(* CODESYS project devicelib.library
   Author: AMKO-Engineering
   Placeholder: Device_Library
   Title: Device_Library
   Version: 1.2.0.3
   Description: Device library of AMKO-Engineering.
   Company: AMKO-Engineering

Project tree, tasks and I/O mapping:
  libraries: HMI_Library, * (AMKO-Engineering); Tc2_MC2, * (Beckhoff Automation GmbH); Tc2_MC2_Drive, * (Beckhoff Automation GmbH); Tc2_Standard, * (Beckhoff Automation GmbH); Utilities_Library, * (AMKO-Engineering)
  Actuators/
    Cylinder/
      DataTypes/
        ManualControls/
          data type UDT_ManualValveControl
        data type E_CylinderCmd
        data type E_ValveResetState
      Functions/
        function block Fb_DevCylWithFbk [ST]: CalcTimers, ExecDirection, ExecSetFeedback, ExecTimeout, CmdSimulate, CmdTeach, Init
        function block FB_DevValve [ST]: ExecSetFeedback, ExecSetOutPuts, CmdClose, CmdHold, CmdManual, CmdOpen, CmdReset, CmdSafeStop, CmdTeach, Init
      MLTFunctions/
        function block Fb_DevSupportCyl [ST]: ExecCalc, ExecCylControl, ExecFaultHandling, Init_Support, Mod_ManualControl, Mod_SupportDown
  Axis/
    DataTypes/
      data type E_AxisCmd
      data type UDT_AxisData
      data type UDT_AxVal
    FunctionBlocks/
      function block Fb_DevAxis [ST]: CmdGearDynamic, CmdGearIn, CmdGearOut, CmdHalt, CmdHome, CmdJog, CmdLimitVelocity, CmdManual, CmdMoveAbs, CmdMoveModulo, CmdMoveRelative, CmdMoveVelocity, CmdReset, CmdSafeSpeed, CmdSafeStop, Init, ExecGearDynamic, ExecGearIn, ExecGearOut, ExecHalt, ExecHome, ExecJog, ExecMoveAbsolute, ExecMoveModulo, ExecMoveRelative, ExecMoveVelocity, ExecEnable, ExecReadStatus, ExecReset, ExecSafeFunctions, CallMotionFunctions, CallOrganizationFunctions
      function block FB_DevBasicACAxis [ST]: CmdHalt, CmdHome, CmdJog, CmdManual, CmdMoveAbs, CmdMoveRelative, CmdMoveVelocity, CmdReset, CmdSafeStop, Init, ExecEnable, ExecHalt, ExecHome, ExecJog, ExecMoveAbsolute, ExecMoveRelative, ExecMoveVelocity, ExecReset, ExecSafeFunctions, CallMotionFunctions
      function block FB_DevHybridAc [ST]: ExecHalt, ExecReadStatus, ExecReset, Init
      data type UDT_ManualAxisCtrl
    Interface/
  BaseFunctions/
    function block FB_DevBase [ST]: ExecIdentifyDevice, CalcDeviceId, CmdManual, CmdReset, CmdSafeStop, ExecMessagTest
    data type UDT_DevManualCtrl
  Buttons/
    DataTypes/
    Functions/
      function block FB_DevHMIButton [ST]
      function block FB_DevPushButton [ST]
      function block FB_DevPushbuttonLight [ST]: CmdBlinkFast, CmdBlinkSlow, CmdOn
  DevTypes/
    data type E_Devices
  Encoders/
    DataTypes/
    FunctionBlocks/
      function block FB_EncoderBase [ST]: FastTask
      function block FB_EncoderInput [ST]: FastTask
  GroupHandlers/
    ManualControlHandler/
      function block FB_ManualController [ST]: ExecSelectDevice, CmdAddDevice
      data type UDT_DeviceID
    global variables GVL_DevManual
  HardwareDiagnostics/
    function block FB_ELModuleDiag [ST]
  Heaters/
    function block FB_DevDoublePWM [ST]: CalcCycleTimes, ExecPWMCycle, SetOutputs, CmdHold, CmdOutputAOn, CmdOutputBOn, CmdSafeStop, Init
    function block FB_DevPWMGenerator [ST]: CalcCycle, ExecSetOutput, CmdOutputCycle, CmdOutputOff, CmdOutputOn
  Lights/
    DataTypes/
    Functions/
      function block Fb_DevLight [ST]: ExecSetOutput, CmdBlinkFast, CmdBlinkSlow, CmdOn
  Outputs/
    AnalogOutputs/
      function block FB_DevAnalogOutput [ST]: ExecSetFeedback, ExecSetOutput
      function block FB_DevAnalogOutputScaled [ST]: ExecSetFeedback, ExecSetOutput, SetScaling
    DigitalOutputs/
      function block FB_DevDigitalOutput [ST]: ExecSetFeedback, ExecSetOutput
  Sensors/
    AnalogInput/
      FunctionBlocks/
        function block FB_DevAnalogInAutoCalibrate [ST]: CmdCalibrateNull, CmdCalilbrateValue
        function block FB_DevAnalogInput [ST]: ExecSetFeedback
        function block FB_DevAnalogInputScaled [ST]: ExecSetFeedback, SetScaling
        function block FB_DevHDAnalogInAutoCalibrate [ST]: CmdCalibrateNull, CmdCalilbrateValue
        function block FB_DevHDAnalogInput [ST]: ExecSetFeedback
        function block FB_DevHDAnalogInputScaled [ST]: ExecSetFeedback, SetScaling
    DigitalSensor/
      DataTypes/
      FunctionBlocks/
        function block Fb_DevDigitalInput [ST]
        function block Fb_DevDigitalInputFunctions [ST]
    FootPedals/
      DataTypes/
        data type E_FootpedalPos
      FunctionBlocks/
        function block FB_EfkaEB301A_FootPedal [ST]: ACT_ConvertGreycode, ACT_CreateEdges
    ModuleSpecific/
      EL3556_Loadcell/
        function block Fb_DevEL3356_LoadCell [ST]: CheckELSignalState, CmdCalibrateNull, CmdCalilbrateValue
  Version/
    global variables Global_Version
*)

// Actuators/Cylinder/DataTypes/ManualControls/UDT_ManualValveControl
TYPE UDT_ManualValveControl extends UDT_DevManualCtrl:
STRUCT
	// Device commands
	bCmdOpen	: BOOL	; // open valve 
	bCmdClose	: BOOL	; // Close valve
	bCmdTeach	: BOOL	; // Teach valve
END_STRUCT
END_TYPE

// Actuators/Cylinder/DataTypes/E_CylinderCmd
(* cylinder commands *)
TYPE E_CylinderCmd :
(
	Cyl_Idle 		:= 0,// Jog Cylinder command Referance 0 Idle (wait for command)
	Cyl_Init 		:= 1,// Jog Cylinder command Referance 1 initialize Cylinder
	Cyl_Enable 		:= 2,// Jog Cylinder command Referance 2 enable
	Cyl_Disable 	:= 3,// Jog Cylinder command Referance 3 disable
	Cyl_Reset 		:= 4,// Jog Cylinder command Referance 4 reset
	Cyl_Hold 		:= 5,// Jog Cylinder command Referance 5 hold
	Cyl_Teach 		:= 6,// Jog Cylinder command Referance 6 teach timeout settings
	Cyl_Calculate 	:= 7,// Jog Cylinder command Referance 7 calculate timeout settings from parameters
	Cyl_Expand 		:= 8,// Jog Cylinder command Referance 8 expand
	Cyl_Retract 	:= 9 // Jog Cylinder command Referance 9 retract
);
END_TYPE

// Actuators/Cylinder/DataTypes/E_ValveResetState
{attribute 'qualified_only'}
{attribute 'strict'}
TYPE E_ValveResetState :
(
	Res_Idle 		:= 0,
	Res_Closed		:= 1,
	Res_Open		:= 2
);
END_TYPE

// Axis/DataTypes/E_AxisCmd
(* axis command structure *)
TYPE E_AxisCmd :
(
	Ax_Idle 		:= 0,// Axis command Referance 0 Axis Idle
	Ax_Init 		:= 1,// Axis command Referance 1 Initialize axis
	Ax_Enable 		:= 2,// Axis command Referance 2 Enable
	Ax_Disable 		:= 3,// Axis command Referance 3 Disable
	Ax_Reset 		:= 4,// Axis command Referance 4 Reset
	Ax_Hold 		:= 5,// Axis command Referance 5 Hold
	Ax_Home 		:= 6,// Axis command Referance 6 Home
	Ax_JogFwd 		:= 7,// Axis command Referance 7 Jog Forward
	Ax_JogRev 		:= 8,// Axis command Referance 8 Jog Reverse
	Ax_MoveRelative := 9,// Axis command Referance 9 Move axis relative
	Ax_MoveAbs 		:= 10,// Axis command Referance 11 Move absolute reverse
	Ax_MoveModulo 	:= 11,// Axis command Referance 11 Move Module
	Ax_MoveVeloFwd 	:= 12,// Axis command Referance 12 Move velocity forward
	Ax_MoveVeloRev 	:= 13,// Axis command Referance 13 Move velocity reverse
	Ax_HardStop 	:= 14,// Axis command Referance 14 hard stop or emergency stop
	Ax_SoftStop 	:= 15,// Axis command Referance 15 soft stop after motion command
	Ax_GearSlave 	:= 16,// Axis command Referance 16 gear axis as slave
	Ax_GearSlaveDyn	:= 17,// Axis command Referance 17 gear axis as slave dynamic
	Ax_GearOutSlave := 18,// Axis command Referance 18 gear out from Master axis 
	Ax_Maintenance	:= 50 // Axis Command referance 50 maintenance mode, axis enabled with no command active
);
END_TYPE

// Axis/DataTypes/UDT_AxisData
TYPE UDT_AxisData:
STRUCT
	// ===== Axis name =====
		AxisName	: STRING 	; // Name of the axis (used for fault handling and identification)
		AxisNumber	: INT		; // Axis number 

	// ===== Fault data =====
		Message			: UDT_Fault 	; // Message data from Cylinder
		MessageActive	: BOOL			; // Message is active
		ErrorActive 	: BOOL 			;	// Axis in error state

	// ===== Axis Commands =====
		// ***** Enable command	*****
			CmdEnable		: BOOL 		; // Command enable axis
		// ***** Active commands *****
			AxisCmd			: E_AxisCmd ; // Axis command
			AxisSafeCmd		: E_AxisCmd	; // Axis safe command
			AxisAct			: E_AxisCmd ; // Axis Active status
		// ***** Command Modes *****
			CmdHomingMode 	: MC_HomingMode ; // Homing Mode ( MC_DefaultHoming, MC_Direct, MC_ForceCallibration, MC_ResetCallibration)
			CmdJogMode		: E_JogMode 	;
			CmdBuffermode	: MC_BufferMode	; // Buffermode used for command transition 	 
	// ===== Axis Safe commands =====
		SafeCmdLimitVelo: BOOL 	; // safe command limit velocity
		SafeCmdVelocity	: LREAL ; // Safe command velocity
		SafeCmdStop		: BOOL 	; // Stop command from safety or collision detection		
		SafeVeloLimit	: LREAL ; // safe velocity limit (link to FPAR)
	// ===== Status indication active =====
		ActHoming	: BOOL ; // Axis is homing
		ActBusy		: BOOL ; // Axis is Busy 
		ActMoving	: BOOL ; // Axis is moving
		ActAtVelo	: BOOL ; // Axis is at command velocity (only when written in Move velocity mode)

	// ===== Status indication done  =====
		FcoInit		: BOOL ; // Axis is initialised
		FcoIdle		: BOOL ; // Axis is idle enable required
		FcoEnabled	: BOOL ; // Axis is enabled
		FcoHomed	: BOOL ; // Axis is homed
		FcoGeared	: BOOL ; // Axis is geared to master axis
		FcoHeld		: BOOL ; // Axis is holding
		FcoStopped	: BOOL ; // Axis is stopped
		FcoReset	: BOOL ; // Axis reset done
		FcoReady 	: BOOL ; // Axis is ready for command
		FcoAtCmdPos	: BOOL ; // Axis is at command position (tol 0.2 deg)
		FcoCmdActive: BOOL ; // Axis new command values are active
		
	// ===== Move values =====
		Pos			: UDT_Axval	; // possition values (0 = infinite)
		Velocity 	: UDT_AxVal	; // Velocity values
		Accel		: UDT_Axval ; // Aceleration values
		Decel		: UDT_Axval ; // Deceleration values
		Torque		: UDT_Axval ; // Torque values
		EncTurnoverVal	: DINT 	; // Encoder turnover value
		TimeDisableDelay : TIME ; // Time off delay after axis move command (remove enable)
		
	// ===== Config Bits =====
		IcfCommandSpeedRpm	: BOOL ; // input speeds in Rpm
		IcfEnableForward 	: BOOL ; // Enable forward motion
 		IcfEnablereverse	: BOOL ; // Enable reverse motion
		IcfContinuous		: BOOL ; // continuous motion possible (no endpoint)
		IcfAlwaysEnable		: BOOL ; // 1 = Axis always enabled, 0 = Axis disabled at Idle 
		
	// ===== Master Axis =====
		MasterAxisRef	: REFERENCE TO AXIS_REF ; // Master axis reference (if applicable)
		GearMasterRev	: UINT	:= 1	; // Master Axis Gearing revolutions (Denominator)
		GearSlaveRev	: LREAL	:= 1	; // Slave Axis gearing revolutions (numerator)	
		ReverseSlave	: BOOL 	; // Reverse slave axis relative to master
		 
END_STRUCT
END_TYPE

// Axis/DataTypes/UDT_AxVal
TYPE UDT_AxVal :
STRUCT
	// ***** Velocity settings *****
		HardMax		: LREAL 	; // Hardware maximum set absolute maximum
		ManMax 		: LREAL		; // Manual maximum percentage of hardware max
		AutoMax		: LREAL		; // Automatic maximum percentage of hardware max
		HomeMax		: LREAL 	; // Homing maximum percentage of hardware max
		CmdVal		: LREAL 	; // Commanded value
		SafeVal		: LREAL		; // Command value after safety check
		PrevVal		: LREAL		; // previous command value 
		ActVal		: LREAL		; // Actual value
		ActModulo	: LREAL		; // [deg] Modulo position
		RefVal		: LREAL 	; // referance value (basic setting or home) 
END_STRUCT
END_TYPE

// Axis/FunctionBlocks/UDT_ManualAxisCtrl
TYPE UDT_ManualAxisCtrl :
STRUCT
	bCmdJogForward	: 	BOOL 		; // command jog forward
	bCmdJogReverse	: 	BOOL 		; // command jog reverse
	bCmdInching		: 	BOOL 		; // Command move relative Distance
	bCmdToPos		: 	BOOL 		; // command move to absolute position (only moving when active)
	bCmdHome		: 	BOOL 		; // Command home axis
	fPosition		:	LREAL 		; // target position
	fDistance		:	LREAL 		; // target position
	fVelocity		: 	LREAL 		; // Maximum velocity [units/sec]
END_STRUCT
END_TYPE

// BaseFunctions/UDT_DevManualCtrl
TYPE UDT_DevManualCtrl :
STRUCT
END_STRUCT
END_TYPE

// DevTypes/E_Devices
{attribute 'qualified_only'}
{attribute 'strict'}
{attribute 'To String'}
TYPE E_Devices :
(
	Undefined,
	Valve,
	Cylinder,
	Axis,
	PushButtonLight,
	DigitalSensor,
	AnalogSensor,
	DigitalOut,
	AnalogOut,
	PWMController,
	DoublePWMController	
)INT;
END_TYPE

// GroupHandlers/ManualControlHandler/UDT_DeviceID
TYPE UDT_DeviceID :
STRUCT
	sName			: STRING	; // device name
	sType			: STRING	; // Type of device [string for visu]
	pFunction		: POINTER TO FB_DevBase ; // Pointer to the device
END_STRUCT
END_TYPE

// Sensors/FootPedals/DataTypes/E_FootpedalPos
{attribute 'qualified_only'}
{attribute 'strict'}
TYPE E_FootpedalPos :
(
	eReverse2 	,
	eReverse1 	,
	eIdle		,
	eForward1	,
	eForward2	,
	eForward3	,
	eForward4	,
	eForward5	,
	eForward6	,
	eForward7	,
	eForward8	,
	eForward9	,
	eForward10	,
	eForward11	,
	eForward12	,
	eForward13	,
	eFalse			
) INT; 
END_TYPE

// GroupHandlers/GVL_DevManual
{attribute 'qualified_only'}
VAR_GLOBAL
	fbManualControler	: FB_ManualController ; // Default Manual control function for devices (not called implicitly) 
	bManualModeActive	: BOOL ; // System manual mode is active
END_VAR
VAR_GLOBAL CONSTANT
	nMAXDEVCOUNT		: UDINT  := 100		; // Maximum number of devices 
END_VAR

// Version/Global_Version
{attribute 'TcGenerated'}
{attribute 'no-analysis'}
{attribute 'linkalways'}
// This function has been automatically generated from the project information.
VAR_GLOBAL CONSTANT
	{attribute 'const_non_replaced'}
	stLibVersion_Device_Library : ST_LibVersion := (iMajor := 1, iMinor := 2, iBuild := 0, iRevision := 3, nFlags := 0, sVersion := '1.2.0.3');
END_VAR

// Actuators/Cylinder/Functions/Fb_DevCylWithFbk
FUNCTION_BLOCK PUBLIC Fb_DevCylWithFbk EXTENDS FB_DevValve
VAR_INPUT
	bIcfFbkOpenPresent 	: BOOL := FALSE ; // Feedback for cylinder open is present 
	bIcfFbkClosedPresent: BOOL := FALSE ; // Feedback for Cylinder closed is present
	bIcfTimeChecked		: BOOL := TRUE 	; // Cylinder timing is checked = default true
	nMargin				: LREAL:= 10	; // % of tollerance in move speed 
END_VAR
VAR_OUTPUT
	// ===== Teach function =======
	bCmdCopyTimeParam 	: BOOL	:= FALSE 	;// Cylinder, Command to higher level copy toucht time to parameters
	bFeClosed			: BOOL 	:= FALSE	; // closed sensor falling edge
	bReClosed			: BOOL 	:= FALSE	; // closed sensor rising edge
	bFeOpen				: BOOL 	:= FALSE 	; // Open sensor falling edge
	bReOpen				: BOOL 	:= false 	; // open sensor rising edge 
END_VAR
VAR	
	bFcoCalcDone	: BOOL := FALSE ; // Calculate timers done 
	
	stTimesClose	: Udt_TimerBandwith ; // Timer bandwith for cylinder close
	stTimesOpen		: Udt_TimerBandwith	; // Timer bandwitch for cylinder open 
	
	fbSensorClosed	: Fb_DevDigitalInputFunctions ; // Digital sensor function closed detection
	fbSensorOpen	: Fb_DevDigitalInputFunctions ; // Digital sensor function open detection
	
	fbTimerOpen		: TON ; // Timer for cylinder to open
	fbTimerClose 	: TON ; // Timer for cylinder to close
	fbTimerTeach	: TON ; // timer for teachin cylinder 

	rtCmdWriteParam	: R_TRIG ; // Write parameter rising edge trigger 
	// Simulation
	fbTimerSimOpen 	: TON 	; 
	fbTimerSimClose	: TON 	; 
	
	// Time Cylinder valid 
	bTriggerTimeClose	: BOOL ;
	bTriggerTimeOpen	: BOOL ;
END_VAR

// set device type
	IF eDevType = E_Devices.Undefined THEN 
		eDevType := E_Devices.Cylinder ;
	END_IF

// call base function 
	SUPER^();

// check for device init
	IF NOT bInitOk THEN
		RETURN;
	END_IF 

// ====== Check direction of movement =======
	ExecDirection();
	
// ====== Check movement speed =======
	ExecTimeout();
	
// ====== Calculate timers =======
	CalcTimers();

METHOD PRIVATE CalcTimers : BOOL
VAR
END_VAR
IF stParTimeToClose.fValue = stTimesClose.Nominal AND stParTimeToOpen.fValue = stTimesOpen.Nominal AND bFcoCalcDone THEN 
	RETURN ;
ELSE
	bFcoCalcDone := FALSE ;
END_IF
 
// ====== Calculate close times ======
	stTimesClose.Nominal 	:= stParTimeToClose.fValue ;
	stTimesClose.Maximum 	:= stParTimeToClose.fValue * (1 + (nMargin / 100));
	stTimesClose.Minimal 	:= stParTimeToClose.fValue * (1 - (nMargin / 100));

// ====== Calculate open times ======
	stTimesOpen.Nominal 	:= stParTimeToOpen.fValue ;
	stTimesOpen.Maximum 	:= stParTimeToOpen.fValue * (1 + (nMargin / 100));
	stTimesOpen.Minimal 	:= stParTimeToOpen.fValue * (1 - (nMargin / 100));
	
// ====== Set feedback =======
	bFcoCalcDone := TRUE ;

// ===== send write parameters command ======	
	rtCmdWriteParam(CLK := bFcoCalcDone);
	bCmdCopyTimeParam := rtCmdWriteParam.Q	;
END_METHOD

METHOD PRIVATE ExecDirection : BOOL
VAR_INPUT
END_VAR
// ===== Check direction commands =====
 	IF q_Close AND fbSensorOpen.bReStatus AND NOT q_Open THEN
		stFault.Active			:= TRUE ;
		stFault.MessageNumber	:= E_MessageNumbers.CF_WrongDirection 	;
		stFault.Discription		:= CONCAT( sDevName,'Cylinder Opening instead of closing');
		stFault.FaultType		:= E_FaultTypes.CF 					;
		bErrorActive			:= TRUE 								;
		refFbFault.CmdAddFault( stFault );
	ELSIF q_Open AND fbSensorClosed.bReStatus AND NOT q_close THEN
		stFault.Active			:= TRUE ;
		stFault.MessageNumber	:= E_MessageNumbers.CF_WrongDirection 	;
		stFault.Discription		:= CONCAT( sDevName,'Cylinder closing instead of opening');
		stFault.FaultType		:= E_FaultTypes.CF 					;
		bErrorActive			:= TRUE 								;
	END_IF
END_METHOD

METHOD PROTECTED ExecSetFeedback : BOOL
VAR_INPUT
END_VAR
// ====== Call sensor Open function =======
	IF bIcfFbkClosedPresent THEN 
		fbSensorClosed();
		bFco_Closed := fbSensorClosed.bFcoInputActive ;
		bFeClosed 	:= fbSensorClosed.bFeStatus ;
		bReClosed 	:= fbSensorClosed.bReStatus ;
	ELSE 
		fbTOnClose	(IN 	:= q_Close, PT 	:= LREAL_TO_TIME(stParTimeToClose.fValue))	;
		bFco_Closed := fbTOnClose.Q ;
	END_IF

// ====== Call sensor Close function =======
	IF bIcfFbkOpenPresent THEN 
		fbSensorOpen() 	;
		bFco_open 	:= fbSensorOpen.bFcoInputActive ;
		bFeOpen		:= fbSensorOpen.bFeStatus;
		bReOpen		:= fbSensorOpen.bReStatus;
	ELSE 
		FbTOnOpen	(IN 	:= q_Open, PT 	:= LREAL_TO_TIME(stParTimeToOpen.fValue))	;
		bFco_Open := FbTOnOpen.Q ;
	END_IF

// ====== set outputs =======
	bReady		:= bFco_Closed OR bFco_Open ;
END_METHOD

METHOD PRIVATE ExecTimeout : BOOL
VAR_INPUT
END_VAR
VAR
	nTimePassedMs : LREAL ;
END_VAR
IF bFcoCalcDone AND bIcfTimeChecked AND bEnable THEN 
// ====== Set triggers ======
	IF q_Close  AND bFco_Open THEN 
		bTriggerTimeClose := TRUE ;
	ELSIF q_Open OR bFco_Closed  THEN 
		bTriggerTimeClose := FALSE ;
	END_IF

	IF q_Open  AND bFco_Closed THEN 
		bTriggerTimeOpen := TRUE ;
	ELSIF q_Close OR bFco_Open THEN
		bTriggerTimeOpen := FALSE ;
	END_IF
ELSE
	bTriggerTimeClose 	:= FALSE ;
	bTriggerTimeOpen	:= FALSE ;
END_IF


//======= run timers =======
	IF bIcfFbkClosedPresent THEN 
		fbTimerClose(IN := q_Close AND bEnable, PT := T#1M);
	END_IF	
	
	IF bIcfFbkOpenPresent THEN 
		fbTimerOpen	(IN := q_Open AND bEnable , PT := T#1M);
	END_IF

//====== Run timeout checks for cylinder close =======
	nTimePassedMs:= TIME_TO_LREAL(fbTimerClose.ET);
	
	IF bIcfFbkClosedPresent THEN 
		IF bTriggerTimeClose THEN 
			IF fbSensorClosed.bReStatus THEN 
				IF nTimePassedMs < stTimesClose.Minimal THEN 
					stFault.Active			:= TRUE 							;
					stFault.MessageNumber	:= E_MessageNumbers.CF_MoveToFast 	;
					stFault.Discription		:= CONCAT( sDevName,'Cylinder closing to fast')		;
					stFault.FaultType		:= E_FaultTypes.CF 					;
					bErrorActive			:= TRUE 							;
				END_IF
			ELSIF	nTimePassedMs > stTimesClose.Maximum  THEN
				stFault.Active			:= TRUE ;
				stFault.MessageNumber	:= E_MessageNumbers.CF_MoveToSlow 	;
				stFault.Discription		:= CONCAT( sDevName,'Cylinder closing to Slow')		;
				stFault.FaultType		:= E_FaultTypes.CF 				;
				bErrorActive			:= TRUE 							;
			END_IF
		END_IF
	END_IF	

//====== Run timeout checks for cylinder Open =======
	nTimePassedMs:= TIME_TO_REAL(fbTimerOpen.ET);

	IF bIcfFbkOpenPresent THEN 
		IF bTriggerTimeOpen THEN 
			IF fbSensorOpen.bReStatus THEN 
				IF nTimePassedMs < stTimesOpen.Minimal THEN 
					stFault.Active			:= TRUE ;
					stFault.MessageNumber	:= E_MessageNumbers.CF_MoveToFast 	;
					stFault.Discription		:= CONCAT( sDevName, 'Cylinder Opening to fast'	)	;
					stFault.FaultType		:= E_FaultTypes.CF 				;
					bErrorActive			:= TRUE 							;
				END_IF
			ELSIF	nTimePassedMs > stTimesOpen.Maximum  THEN
				stFault.Active			:= TRUE ;
				stFault.MessageNumber	:= E_MessageNumbers.CF_MoveToSlow 	;
				stFault.Discription		:= CONCAT( sDevName,'Cylinder Opening to Slow')		;
				stFault.FaultType		:= E_FaultTypes.CF 				;
				bErrorActive			:= TRUE 							;
			END_IF
		END_IF
	END_IF	

// Handle faults 
IF stFault.Active THEN 
	refFbFault.CmdAddFault( stFault );
END_IF
END_METHOD

METHOD PUBLIC CmdSimulate : BOOL
VAR_INPUT
	bFbkReverse		: BOOL := FALSE ; 
	tTimeSimOpen	: TIME := T#1S 	;
	tTimeSimClose	: TIME := T#1S 	;  
END_VAR
// Run timers when cylinder is active 
	fbTimerSimOpen	(IN := q_Open	, PT := tTimeSimOpen);
	fbTimerSimClose	(IN := q_Close	, PT := tTimeSimClose);

// set feedback sensors to simulate
	fbSensorOpen.bCmdSimulate 	:= TRUE ;
	fbSensorClosed.bCmdSimulate := TRUE ;

// set simulated feedback state 
	IF bFbkReverse THEN 
		fbSensorClosed.bSimState:= fbTimerSimOpen.Q 	;
		fbSensorOpen.bSimState	:= fbTimerSimClose.Q 	; 	
	ELSE 
		fbSensorClosed.bSimState:= fbTimerSimClose.Q 	;
		fbSensorOpen.bSimState	:= fbTimerSimOpen.Q 	; 	
	END_IF
END_METHOD

METHOD PUBLIC CmdTeach : BOOL
VAR_INPUT
END_VAR
// ====== turn off time check function until new calculation cycle =======
	bFcoCalcDone := false ;

// ====== teach cylinder from hardware inputs ======
	fbTimerTeach	(PT:= T#60S);
	fbTimerSwitchDir(PT:= T#1S); 
// ====== time cylinder cycles ======
	// ===== Start test loop =====
	IF bFco_Closed AND fbTimerSwitchDir.Q THEN
		bCmdClose 			:= FALSE;
		bCmdOpen 			:= TRUE ;
		fbTimerSwitchDir.IN	:= FALSE; 
		fbTimerTeach.IN 	:= TRUE ;
	ELSIF bFco_Open AND fbTimerSwitchDir.Q THEN
		bCmdClose 			:= TRUE ;
		bCmdOpen 			:= FALSE;
		fbTimerSwitchDir.IN	:= FALSE; 
		fbTimerTeach.IN 	:= TRUE ;
	ELSIF NOT bCmdClose AND NOT bCmdOpen THEN 
		bCmdClose 			:= TRUE ;
		bCmdOpen 			:= FALSE;
		fbTimerTeach.IN 	:= TRUE ;
	END_IF

// ====== start timing ========
	IF bCmdClose AND bFco_Closed THEN 
		IF fbTimerTeach.IN THEN
			stParTimeToClose.fValue 	:= TIME_TO_LREAL(fbTimerTeach.ET);
		END_IF
		fbTimerSwitchDir.IN := TRUE 		;
		fbTimerTeach.IN 	:= FALSE 		;
	ELSIF bCmdOpen AND bFco_Open THEN 
		IF fbTimerTeach.IN THEN
			stParTimeToOpen.fValue		:= TIME_TO_LREAL(fbTimerTeach.ET);
		END_IF
		fbTimerSwitchDir.IN := TRUE 		;
		fbTimerTeach.IN 	:= FALSE 		;
	END_IF
END_METHOD

METHOD PUBLIC Init : BOOL
VAR_INPUT
	// Valve data
	nDevNumber	: UDINT				:= 0		; // Cylinder identification number
	// Command state
	eResetState		: E_ValveResetState := 0		; // Cylinder reset state variable (default is idle) 
	eSafeState		: E_ValveResetState	:= 0		; // Valve safe state
END_VAR
bFcoCalcDone := FALSE;

// Enable sensor feedback
fbSensorClosed.bEnable	:= TRUE ;
fbSensorOpen.bEnable	:= TRUE ;

// Call feedback sensors 
ExecSetFeedback(); 

SUPER^.Init(nDevNumber, eResetState, eSafeState);

// ===== Set device type for manual control =====
eDevType := E_Devices.Cylinder ;


Init := bInitOk ;
END_METHOD

END_FUNCTION_BLOCK

// Actuators/Cylinder/Functions/FB_DevValve
FUNCTION_BLOCK PUBLIC FB_DevValve EXTENDS FB_DevBase
VAR_INPUT
	// Manual control 
	stManualCtrl	: UDT_ManualValveControl ;
END_VAR
VAR_OUTPUT
	// ===== Status indicators =======
	bFco_Closed		:	BOOL := FALSE ;
	bFco_Open		: 	BOOL := FALSE ;
END_VAR
VAR
	// Pararmeters
		stParTimeToClose	: Udt_Parameter := (fValue := 50) ; // time to close parameter
		stParTimeToOpen		: Udt_Parameter	:= (fValue := 50) ; // Time to open parameter
	// Hardware links 
		q_Open			AT %Q* : BOOL := FALSE 	; // Open valve
		q_Close 		AT %Q* : BOOL := FALSE	; // Close valve
	// Internal commands
		bCmdClose 	: BOOL := FALSE ; // close valve 
		bCmdOpen	: BOOL := FALSE ; // Open valve
		bCmdHold	: BOOL := FALSE ; // Hold valve status change
	// Time functions 
		fbTOnClose	: TON	; // Timer for valve close
		FbTOnOpen	: TON 	; // Timer for valve Open
		fbTimerSwitchDir: TON ; // Time for teach function switch direction 
	// reset and safe state
		eResetState		: E_ValveResetState := 0		; // Cylinder reset state variable (default is idle) 
		eSafeState		: E_ValveResetState	:= 0		; // Valve safe state
END_VAR

// set device type
IF eDevType = E_Devices.Undefined THEN 
	eDevType := E_Devices.Valve ;
END_IF

// Call base function
SUPER^();

// ===== hold all actions if not initialized ======
IF NOT bInitOk THEN
	RETURN;
END_IF 

// ====== Set Outputs =======
	ExecSetOutPuts();

// ===== collect feedback ======
	ExecSetFeedback();

METHOD PROTECTED ExecSetFeedback : BOOL
VAR_INPUT
END_VAR
// ====== Set timers =======
	fbTOnClose	(PT 	:= LREAL_TO_TIME(stParTimeToClose.fValue))	;
	FbTOnOpen	(PT		:= LREAL_TO_TIME(stParTimeToOpen.fValue))	;

// ====== Set timed feedback ======
	IF q_Close THEN 
		fbTOnClose.IN 	:= TRUE ;
		fbTOnopen.IN 	:= FALSE;
	ELSIF q_Open THEN 
		fbTOnClose.IN 	:= FALSE;
		FbTOnOpen.IN	:= TRUE ;
	ELSE 
		fbTOnClose.IN 	:= FALSE;
		FbTOnOpen.IN	:= FALSE;
	END_IF
	
// ====== set outputs =======
	bFco_Closed := fbTOnClose.Q ;
	bFco_Open	:= FbTOnOpen.Q	;
	bReady		:= bFco_Closed OR bFco_Open ;
END_METHOD

METHOD PROTECTED ExecSetOutPuts : BOOL
VAR_INPUT
END_VAR
// ======= Set Outputs according to commands and check safety features =======
IF bSafetyOk THEN
	IF NOT bCmdHold AND (bEnable OR bCmdManual) THEN  
		q_Close	:= bCmdClose;
		q_Open	:= bCmdOpen	;
		bBlockedCommand := FALSE ;
	ELSE
		bBlockedCommand := TRUE ;
	END_IF
ELSE
	CASE eSafeState OF 
		E_ValveResetState.Res_Idle:
			q_Close	:= bFco_Closed;		
			q_Open 	:= bFco_Open;
		E_ValveResetState.Res_Closed:
			q_Close	:= TRUE	;		
			q_Open 	:= FALSE;
		E_ValveResetState.Res_Open:
			q_Close	:= FALSE;		
			q_Open 	:= TRUE	;
	END_CASE
	bCmdClose 	:= bFco_Closed 	;
	bCmdOpen	:= bFco_Open	;
	
END_IF

// Reset manual and hold commands
bCmdHold 	:= FALSE ;
bCmdManual 	:= FALSE ;
END_METHOD

METHOD PUBLIC CmdClose : BOOL // close valve or retract cylinder
VAR_INPUT
END_VAR
// ====== Set close command if enabled ======
	bCmdClose 	:= TRUE	;		
	bCmdOpen 	:= FALSE;
	
// ===== Set feedback ======
	CmdClose := bFco_Closed ;
END_METHOD

METHOD PUBLIC CmdHold : BOOL
VAR_INPUT
END_VAR
// ====== set hold command =====
	bCmdHold := TRUE ;

CmdHold := bBlockedCommand ;
END_METHOD

METHOD PUBLIC CmdManual : BOOL
VAR_IN_OUT
END_VAR
// Enable manual commands
bCmdManual S= TRUE ;

// execute manual command 
	IF stManualCtrl.bCmdOpen THEN 
		CmdOpen();
	ELSIF stManualCtrl.bCmdClose THEN 
	 	CmdClose(); 
	ELSIF stManualCtrl.bCmdTeach THEN
		CmdTeach ();
	END_IF
END_METHOD

METHOD PUBLIC CmdOpen : BOOL // Open valve or retract cylinder
VAR_INPUT
END_VAR
// ====== Set open command if enabled ======
	bCmdClose 	:= FALSE;		
	bCmdOpen 	:= TRUE	;
	
// ===== Set feedback ======
	CmdOpen := bFco_Open ;
END_METHOD

METHOD CmdReset : BOOL
VAR_INPUT
END_VAR
// ====== Set outputs according to reset state =======
	IF bEnable THEN 
		CASE eResetState OF 
			E_ValveResetState.Res_Idle:
				bCmdClose 	:= FALSE;		
				bCmdOpen 	:= FALSE;
			E_ValveResetState.Res_Closed:
				bCmdClose 	:= TRUE	;		
				bCmdOpen 	:= FALSE;
			E_ValveResetState.Res_Open:
				bCmdClose 	:= FALSE;		
				bCmdOpen 	:= TRUE	;
		ELSE
			;
		END_CASE
	END_IF
// ======= Reset Error bit ======
	bErrorActive 	:= FALSE;
	bBussy			:= FALSE;
END_METHOD

METHOD PUBLIC CmdSafeStop : BOOL
VAR_INPUT
END_VAR
CASE eSafeState OF 
	E_ValveResetState.Res_Idle:
		bDevIsSafe := bFco_Closed OR bFco_Open ;
	E_ValveResetState.Res_Closed:
		bDevIsSafe := bFco_Closed ;
	E_ValveResetState.Res_Open:
		bDevIsSafe := bFco_Open ;
END_CASE

CmdSafeStop := bDevIsSafe OR NOT bInitOk ;
END_METHOD

METHOD PUBLIC CmdTeach : BOOL
VAR_INPUT
END_VAR
// ====== teach cylinder from hardware inputs ======
	fbTimerSwitchDir(PT:= T#1S); 
// ===== Start test loop =====
IF bFco_Closed AND fbTimerSwitchDir.Q THEN
	bCmdClose 			:= FALSE;
	bCmdOpen 			:= TRUE ;
	fbTimerSwitchDir.IN	:= FALSE; 
ELSIF bFco_Open AND fbTimerSwitchDir.Q THEN
	bCmdClose 			:= TRUE ;
	bCmdOpen 			:= FALSE;
	fbTimerSwitchDir.IN	:= FALSE; 
ELSIF NOT bCmdClose AND NOT bCmdOpen THEN 
	bCmdClose 			:= TRUE ;
	bCmdOpen 			:= FALSE;
END_IF

// ====== start timing ========
	IF bCmdClose AND bFco_Closed THEN 
		fbTimerSwitchDir.IN := TRUE 		;
	ELSIF bCmdOpen AND bFco_Open THEN 
		fbTimerSwitchDir.IN := TRUE 		;
	END_IF
END_METHOD

METHOD PUBLIC Init : BOOL
VAR_INPUT
	// Valve data 
	nDevNumber	: UDINT				:= 0		; // Cylinder identification number
	// Command state
	eResetState		: E_ValveResetState := 0		; // Cylinder reset state variable (default is idle) 
	eSafeState		: E_ValveResetState	:= 0		; // Valve safe state
END_VAR
// ====== Calculate device id =====
	THIS^.nDevNumber := nDevNumber ;
	SUPER^.CalcDeviceId();
// ====== Set message information =======
	stFault.ComponentType	:= E_ComponentTypes.Cylinder 		;
	
// ====== Set outputs according to reset state =======
	THIS^.eResetState 	:= eResetState 	;
	THIS^.eSafeState	:= eSafeState	;	

	IF bEnable THEN 
		CASE eResetState OF 
			E_ValveResetState.Res_Idle:
				bCmdClose 	:= bFco_Closed	;		
				bCmdOpen 	:= bFco_Open	;
			E_ValveResetState.Res_Closed:
				bCmdClose 	:= TRUE;		
				bCmdOpen 	:= FALSE;
			E_ValveResetState.Res_Open:
				bCmdClose 	:= FALSE;		
				bCmdOpen 	:= TRUE ;
		END_CASE
	END_IF
// ======= Reset Error bit ======
	bErrorActive 	:= FALSE;
	bBussy			:= FALSE;

// ===== Set device type for manual control =====
	eDevType := E_Devices.Valve ;
	
// ===== configure parameters =====
	stParTimeToClose.fMinimum 		:= 0 		;
	stParTimeToClose.fMaximum		:= 60000 	;
	stParTimeToClose.nNumber 		:= nDevId + 1;
	stParTimeToClose.sDiscription  	:= CONCAT( STR1 := sDevName, STR2 := 'avarage time it takes for the valve to close in miliseconds');
	stParTimeToClose.sName			:= CONCAT( STR1 := sDevName, STR2 := 'time to close');
	stParTimeToClose.sType			:= 'CPar';
	stParTimeToClose.sUnit			:= 'ms';

	stParTimeToOpen.fMinimum 		:= 0 		;
	stParTimeToOpen.fMaximum		:= 60000 	;
	stParTimeToOpen.nNumber 		:= nDevId + 2;
	stParTimeToOpen.sDiscription  	:= CONCAT( STR1 := sDevName, STR2 := 'avarage time it takes for the valve to open in miliseconds');
	stParTimeToOpen.sName			:= CONCAT( STR1 := sDevName, STR2 := 'time to open');
	stParTimeToOpen.sType			:= 'CPar';
	stParTimeToOpen.sUnit			:= 'ms';
	
	// add parameters to handler 
	refFbParHandler.CmdAddParameter( refParameter := stParTimeToClose );
	refFbParHandler.CmdAddParameter( refParameter := stParTimeToOpen );
	
// ====== Set init status bit =======
	bInitOk := TRUE ;
END_METHOD

END_FUNCTION_BLOCK

// BaseFunctions/FB_DevBase
{attribute 'reflection'}
FUNCTION_BLOCK PUBLIC FB_DevBase
VAR_INPUT
	nModuleId		: UDINT		:= 	1 					; // Higher level module ID
	bEnable			: BOOL 		:= TRUE 				; // Module enable signal reference Default := TRUE (when using system library := GVL_Main.stModules[nModuleId].bEnabled)
	bSafetyOk		: BOOL 		:= TRUE 				; // Module can operate safely [default true]
	bReset 			: BOOL 		:= FALSE				; // reset command bit reference Default := TRUE (when using system library := GVL_Main.stModules[nModuleId].bResetting)
	refFbFault		: REFERENCE TO Fb_FaultHandler	 	; // reference to fault handler ( when using utilities library := GVL_Main.stModules[nModuleId].fbFaultHandler)
	// function references 
	refFbManualCtrl	: REFERENCE TO FB_ManualController := GVL_DevManual.fbManualControler	; // reference to manual handler
	refFbParHandler	: REFERENCE TO Fb_ParLogging 	:= GVL_Parameters.fbParameterHandler	; // reference to parameter handler
END_VAR
VAR_IN_OUT
END_VAR
VAR_OUTPUT
	sDevActiveState	: STRING 		:= 'Idle'	; // active state of device 
	bInitOk			: BOOL 			:= FALSE 	; // function is initialized
	bBussy 			: BOOL 			:= FALSE 	; // device is busy
	bReady			: BOOL 			:= FALSE 	; // device is ready for new command 
	bManual			: BOOL 			:= false 	; // device is in manual mode
	bDevIsSafe		: BOOL 			:= FALSE	; // Device is locked and safe
	bErrorActive	: BOOL			:= FALSE	; // device Error active 
	bBlockedCommand	: BOOL 			:= False 	; // a device command is blocked because of collision detect 
	sDevName		: STRING 		; // Name of device distilled from the path 
	eDevType		: E_Devices	:= E_Devices.Undefined	; // Type of Device 	
	nDevNumber		: UDINT 		:= 0 		; // device sub number
	nDevId			: UDINT 		:= 0		; // device id number made up of module and device number				
END_VAR
VAR
	// Feedback request
	bMessageTest	: BOOL  		:= FALSE	; // Send test message from device
	// ===== Fault data =====
	stFault			: UDT_Fault	; // Fault data from device
	// Manual control variables
	bAddedToManual	: BOOL 			:= FALSE 	; // device is added tot manual control function 	
	bCmdManual 		: BOOL			:= FALSE	; // manual commands enabled control functions (thus disable automatic)
	// Function path 
	{attribute 'instance-path'} 
    {attribute 'noinit'}
	sPath			: STRING	; // Path name of function (used for manual reference)
END_VAR

ExecIdentifyDevice();

// Communicate active state
IF NOT bSafetyOk THEN 
	sDevActiveState := 'Safety not ok';
ELSIF bErrorActive THEN 
	sDevActiveState := TO_STRING(stFault.Discription);
ELSIF NOT bInitOk THEN 
	sDevActiveState := 'Not initialized';
ELSIF bManual THEN 
	sDevActiveState := 'Operational';
END_IF 

// Set fault if commands are blocked
IF bBlockedCommand THEN 
	stFault.Active 			:= TRUE ;
	stFault.ComponentType 	:= E_ComponentTypes.Assembly ;
	stFault.Discription		:= CONCAT( STR1 := sDevName, STR2 := 'Movement path is blocked');
	stFault.FaultType		:= E_FaultTypes.MC;
	refFbFault.CmdAddFault( stFault);
END_IF	
// Call reset function 
IF bReset THEN 
	CmdReset();
END_IF

METHOD PRIVATE ExecIdentifyDevice : BOOL
VAR_INPUT
END_VAR
// Check device ID
IF bInitOk AND nDevId = 0 THEN 
	CalcDeviceId();
END_IF

// set message location information
stFault.LocationName	:= sDevName	;	
stFault.LocationNumber	:= nDevId	;

// Get device name from function and add device to manual
IF sDevName = '' THEN 
	sDevName := F_FBNameFromPath(sPath := sPath);
ELSIF NOT bAddedToManual AND eDevType <> E_Devices.Undefined THEN 
	bAddedToManual S= refFbManualCtrl.CmdAddDevice(THIS^);
END_IF

// Call message test function
ExecMessagTest();

bManual := bCmdManual ;
END_METHOD

METHOD PROTECTED CalcDeviceId : BOOL
VAR_INPUT
END_VAR
nDevId := (nModuleId * 10000) + nDevNumber * 100 ;
END_METHOD

METHOD PUBLIC CmdManual : BOOL
VAR_INPUT
END_VAR
bCmdManual := true ;
END_METHOD

METHOD CmdReset : BOOL
VAR_INPUT
END_VAR
END_METHOD

METHOD PUBLIC CmdSafeStop : BOOL
VAR_INPUT
END_VAR
// check if device is safe
bDevIsSafe 	:= NOT bEnable ;
CmdSafeStop := bDevIsSafe ;
END_METHOD

METHOD ExecMessagTest : BOOL
VAR_INPUT
END_VAR
IF bMessageTest THEN 
	stFault.Active 			:= TRUE ;
	stFault.Discription 	:= CONCAT(STR1 := 'This is a test message from: ',STR2 := sDevName);
	stFault.MessageNumber 	:= E_MessageNumbers.OM_MessageTest ;
	stFault.FaultType		:= Utilities_Library.E_FaultTypes.OM ;
	refFbFault.CmdAddFault( stFault );
END_IF
END_METHOD

END_FUNCTION_BLOCK

// GroupHandlers/ManualControlHandler/FB_ManualController
FUNCTION_BLOCK FB_ManualController
VAR_INPUT
	bReset 			: BOOL 		:= FALSE ; // (auto linked) reset selected device 
END_VAR
VAR_OUTPUT
	eDevType		: INT		:= E_Devices.Undefined	; // Selected device type
	bManual			: BOOL 		:= FALSE ; // selected device is in manual state
	bErroractive	: BOOL 		:= FALSE ; // Device error is active
	sDeviceState	: STRING	:= '' 	; // Dselected device fault message
END_VAR
VAR
	nNumberOfDevices	: UDINT := 0 	; // number of devices in manual array 
	
	bManualActive		: BOOL 	:= FALSE ; // Manual control mode is activated
	bDisableManualInputs: BOOL 	:= TRUE 	; // disable device manual inputs
	
	pDevValve			: POINTER TO FB_DevValve				; // Device pointer to valve
	pDevCylinder		: POINTER TO Fb_DevCylWithFbk 			; // Device pointer to cylinder with manual 
	pDevAxis			: POINTER TO Fb_DevAxis 				; // device pointer to Axis 
	pDevPBL				: POINTER TO FB_DevPushbuttonLight		; // Device pointer to puschbutton light
	pDevDigitalInput	: POINTER TO Fb_DevDigitalInputFunctions; // device pointer to digital input
	pDevAnalogInput		: POINTER TO FB_DevAnalogInput			; // Device pointer to analog input
	pDevAnalogOut		: POINTER TO FB_DevAnalogOutput			; // Device pointer to analog output
	pDevDigitalOut		: POINTER TO FB_DevDigitalOutput		; // Device pointer to digital output
	pDevPWMController	: POINTER TO FB_DevPWMGenerator			; // Device pointer to PWM controller
	pDevDoublePWM		: POINTER TO FB_DevDoublePWM			; // Device pointer to Double PWM controller
	
	fbNodevice			: FB_DevBase ;
	stNoDevice			: UDT_DeviceID := (sName := 'No device', sType := TO_STRING(E_Devices.Undefined), pFunction := ADR(fbNodevice)); 
	arDeviceArray		: ARRAY [0..GVL_DevManual.nMAXDEVCOUNT] OF UDT_DeviceID := [stNoDevice]	; // Array of Devices for manual control
	nCmdLookupindex		: UDINT := 0; // Index number in array
	i					: UDINT := 0; // Index pointer to array
END_VAR

GVL_DevManual.bManualModeActive := bManualActive ;
IF bManualActive THEN 
	// insert a device 
	ExecSelectDevice();
END_IF

METHOD PRIVATE ExecSelectDevice : BOOL
VAR_INPUT
END_VAR
// Select active manual device
bDisableManualInputs := NOT arDeviceArray[nCmdLookupindex].pFunction^.bManual ; 
IF bManualActive THEN 
	arDeviceArray[nCmdLookupindex].pFunction^.CmdManual(); 
END_IF

CASE arDeviceArray[nCmdLookupindex].pFunction^.eDevType OF
	E_Devices.Valve			:
		pDevValve 			:= arDeviceArray[nCmdLookupindex].pFunction ;
	E_Devices.Cylinder		:
		pDevCylinder		:= arDeviceArray[nCmdLookupindex].pFunction ;
	E_Devices.Axis 			:
		pDevAxis			:= arDeviceArray[nCmdLookupindex].pFunction ;
	E_Devices.PushButtonLight :
		pDevPBL				:= arDeviceArray[nCmdLookupindex].pFunction ;
	E_Devices.DigitalSensor :
		pDevDigitalInput	:= arDeviceArray[nCmdLookupindex].pFunction ;
	E_Devices.AnalogSensor 	:
		pDevAnalogInput 	:= arDeviceArray[nCmdLookupindex].pFunction ;
	E_Devices.DigitalOut	:
	 	pDevDigitalOut		:= arDeviceArray[nCmdLookupindex].pFunction ;
	E_Devices.AnalogOut		:
		pDevAnalogOut		:= arDeviceArray[nCmdLookupindex].pFunction ;
	E_Devices.PWMController	:
		pDevPWMController	:= arDeviceArray[nCmdLookupindex].pFunction ;
	E_Devices.DoublePWMController :
		pDevDoublePWM		:= arDeviceArray[nCmdLookupindex].pFunction ;
	ELSE
		;
END_CASE

// Set device command 
arDeviceArray[nCmdLookupindex].pFunction^.bReset := bReset ;

// Set device state feedback
bManual 		:= arDeviceArray[nCmdLookupindex].pFunction^.bManual ;
bErroractive	:= arDeviceArray[nCmdLookupindex].pFunction^.bErrorActive ;
sDeviceState	:= arDeviceArray[nCmdLookupindex].pFunction^.sDevActiveState ;

// Set device screen control 
eDevType := arDeviceArray[nCmdLookupindex].pFunction^.eDevType ;
END_METHOD

METHOD PUBLIC CmdAddDevice : BOOL
VAR_INPUT
	refToDevice	: REFERENCE TO FB_DevBase ;
END_VAR
VAR
	bDevAdded	: BOOL ;
END_VAR
// Check if device is not already in the array 
FOR i:= 0 TO nNumberOfDevices DO 
	IF arDeviceArray[i].sName = refToDevice.sDevName THEN 
		bDevAdded := TRUE ;
	END_IF 
END_FOR

// If device is not found add device to the list
IF NOT bDevAdded THEN 
	nNumberOfDevices := LIMIT(0, nNumberOfDevices + 1 ,GVL_DevManual.nMAXDEVCOUNT)	;
	arDeviceArray[nNumberOfDevices].sType 		:= TO_STRING(refToDevice.eDevType)	;
	arDeviceArray[nNumberOfDevices].sName		:= refToDevice.sDevName	;
	arDeviceArray[nNumberOfDevices].pFunction 	:= ADR(refToDevice)		;	
	bDevAdded := TRUE ;
END_IF

CmdAddDevice := bDevAdded ;
END_METHOD

END_FUNCTION_BLOCK

// Axis/FunctionBlocks/Fb_DevAxis
FUNCTION_BLOCK PUBLIC Fb_DevAxis EXTENDS FB_DevBase
VAR_INPUT
	// ===== General Function input =====
		fCmdAcc			: LREAL := 15000;
		fCmdDecc		: LREAL := 15000; 
	// ===== Master Axis =====
		refMasterAxis	: REFERENCE TO AXIS_REF ; // Master axis reference (if applicable)
		bReverseSlave	: BOOL 	:= FALSE; // Reverse slave axis relative to master
		fCmdGearRatio	: LREAL := 1 ; // Gear ratio Master/Slave (1/Ratio) 
	// Manual control reference
		stManualCtrl	: UDT_ManualAxisCtrl ;
END_VAR
VAR_OUTPUT
	// ====== State indications =======
		bHomed			: BOOL 	:= FALSE; 
		bError 			: BOOL 	:= FALSE;
		bStopped		: BOOL 	:= FALSE;
		bGearedAsSlave	: BOOL 	:= FALSE;
		bVelocityLimited: BOOL 	:= FALSE;  
		bIdle			: BOOL 	:= FALSE;
		fVelocity		: LREAL	:= 0	; // Axis velocity [rpm or units/sec] depending on config
		fActPosition	: LREAL := 0	; // Axis actual position [Units] depending on config	
	// ====== axis reference ======
		AxisRef			: AXIS_REF	; // Axis reference to hardware 
	// ====== Axis Settings ======
		fMaxVelo		: LREAL := 0 ; // Axis Maximum velocity
		fMaxAcc			: LREAL := 0 ; // Axis Maximum cceleration
		fMaxDec			: LREAL := 0 ; // axis Maxium deceleration 
	
		fSafeVeloLimit	: LREAL	:= 200; // Safe velocity limit 
		tEnableDelay	: TIME 	:= T#0MS	;
		tDisableDelay	: TIME 	:= T#500MS  ;
	// ==== Axis data ====
		fEncoderTurnoverValue	: LREAL ;   
END_VAR
VAR // Axis configuration 
	// ===== HW Config Bits =====
		bIcfCmdVelocityRpm	: BOOL ; // input speeds in Rpm
		bIcfEnableForward 	: BOOL ; // Enable forward motion
 		bIcfEnablereverse	: BOOL ; // Enable reverse motion
		bIcfAlwaysEnable	: BOOL ; // 1 = Axis always enabled, 0 = Axis disabled at Idle 
		bIcfSimulationMode	: BOOL := FALSE ; // Simulation mode is active [default set to False] 
	// ===== Internal motion values ======
		fHomePosition		: LREAL := 0 ; // set position at homing
	// Command Modes
		mcHomingMode 		: MC_HomingMode := MC_direct ; // Homing Mode ( MC_DefaultHoming, MC_Direct, MC_ForceCallibration, MC_ResetCallibration)
	// Values from system
		McReadSysVelo		: MC_ReadParameter		; // Read Acceleration parameter from drive 
		McReadSysAcc		: MC_ReadParameter		; // Read Acceleration parameter from drive 
		McReadSysDec		: MC_ReadParameter		; // Read Acceleration parameter from drive 
END_VAR
VAR	// ====== Axis enable =====
		bCmdEnableAxis 		: BOOL 	:= FALSE; // Command to enable the axis (External)
		bInternalEnable		: BOOL 	:= FALSE; // internal enable command (turns off after set time, and on at new motion command
		bDelayedEnable		: BOOL 	:= false; // Delayed enable signal for motion commands
		TonMotionEnable		: TON 			; // Timer on for motion command enable
		TofIntAxisEnable	: TOF  			; // Timer off for internal axis enable 
	// Parameter read status 
		Cmd_EnDriveParRead	: BOOL 			; // Enable parameter read 
	// ===== Physical Homing signal =====
		IAxisHome AT %I* 	: BOOL 			; // Axis homing sensor from PLC (if MC_DefaultHoming is used)
END_VAR
VAR	// =============== Motion status functions ================
		fbMcReadAxisStatus	: MC_ReadStatus ;	// Fb for reading axis status	
	// =============== Motion function blocks =================
		fbMcPower 			: MC_Power		;		// FB for enable and override
		fbMcReset 			: MC_Reset		;		// FB to reset axis
		fbSoeReset			: FB_SoEReset	; 		// FB to reset axis hardware
		fbMcHome			: MC_Home		;		// Fb to home Axis
		fbMcStop 			: MC_Stop		;		// FB to stop axis
		fbMcHalt			: MC_Halt		;		// FB to halt axis
		fbMcJog				: MC_Jog		;		// FB to Jog axis
		fbMcMoveVelocity	: MC_MoveVelocity;		// FB to move with specified velocity until Next command is given
		fbMcGearInSlave		: MC_GearIn		;		// FB to gear axis to master 
		fbMcGearInDyn		: MC_GearInDyn	;		// FB to gear axis dynamicly to master
		fbMcGearOutSlave	: MC_GearOut	;		// FB to decouple gearing

	(* PtoP Motion move commands are in arrays so multiple commands can be stacked *) 
		fbMCMoveRelative	: ARRAY [0..1] OF MC_MoveRelative	;		// FB to move relative
		fbMcMoveAbsolute	: ARRAY [0..1] OF MC_MoveAbsolute	;		// FB to move axis (velocity movement)
		fbMcMoveModulo		: ARRAY [0..1] OF MC_MoveModulo		;		// FB to move axis to modulo position
	// ===== Safe commands =====
		bCmdSafeStop	: BOOL ;
		bCmdSafeSpeed	: BOOL ; 
	// ===== Function execute triggers =====
		bExec_Reset			: BOOL := FALSE; // Execute reset
		bExec_Halt			: BOOL := FALSE; // Execute hold
		bExec_Home			: BOOL := FALSE; // Execute Home
		bExec_JogPositive	: BOOL := FALSE; // Execute Jog in positive direction
		bExec_JogNegative	: BOOL := FALSE; // Execute Jog in negative direction
		bExec_MoveVelocity	: BOOL := FALSE; // Execute move velocity
		bExec_GearAsSlave	: BOOL := FALSE; // Execute gear as slave
		bExec_GearSlaveDyn	: BOOL := FALSE; // Execute gear slave dynamic
		bExec_GearOutSlave	: BOOL := FALSE; // execute gear out slave
	// ===== Move ristrictions ======
		bCmdLimitVelocity 	: BOOL := FALSE			; // velocity limiting is active 
		fCmdVelocityLimit	: LREAL:= fSafeVeloLimit; // Maximum velocity limit when velocity limiting is active  
	(* PtoP Motion move commands are in arrays so multiple commands can be stacked *) 
		arExec_MoveRelative	: ARRAY [0..1] OF BOOL ; // Execute move relative
		arExec_MoveAbs		: ARRAY [0..1] OF BOOL ; // Execute move absolute reverse
		arExec_MoveModulo	: ARRAY [0..1] OF BOOL ; // Execute move modulo
END_VAR
VAR
	// ===== Loop variables =====
		i : DINT := 0 ; // For loop increment
END_VAR

// Call base function
SUPER^(refFbFault := refFbFault);

// ==== Check if axis is initiated =====
IF NOT bInitOk THEN 
	RETURN ; 
END_IF

// ===== Execute safe functions =====
	ExecSafeFunctions(); 
	
// ==== Execute organizational functions =====
	CallOrganizationFunctions();

// ==== execute motion functions =====
	CallMotionFunctions();

METHOD PUBLIC CmdGearDynamic : BOOL // Set axis to geared, activates with variable gear ratio until geared out or stopped (if method is no longer called then gear ratio is locked to last value)
VAR_INPUT
	fGearRatio	:	LREAL	:= 1	; // Slave Axis gearing ratio (Master = 1/ fGearRatio = Slave)	
END_VAR
// set blocked command if halt is active 
bBlockedCommand := fbMcHalt.Active ;

// Set command to true 
bExec_GearSlaveDyn 	:= TRUE ;
bInternalEnable		:= TRUE ;

// coppy parameters
fCmdGearRatio 				:= fGearRatio ;

// Set feedback output 
CmdGearDynamic := fbMcGearInDyn.Active ;
END_METHOD

METHOD PUBLIC CmdGearIn : BOOL // Set axis to geared, activates with constant gear ratio until geared out or stopped
VAR_INPUT
	fGearRatio	:	LREAL	:= 1	; // Slave Axis gearing ratio (Master = 1/ fGearRatio = Slave)	
END_VAR
// set blocked command if halt is active 
bBlockedCommand := fbMcHalt.Active ;

// Set command to true 
bExec_GearAsSlave 	:= TRUE ;
bInternalEnable		:= TRUE ;

// coppy parameters
fCmdGearRatio 				:= fGearRatio ;

// Set feedback output 
CmdGearIn := fbMcGearInSlave.Active ;
END_METHOD

METHOD CmdGearOut : BOOL
VAR_INPUT
END_VAR
// set blocked command if halt is active 
bBlockedCommand := fbMcHalt.Active ;

// Set command to true
bExec_GearOutSlave := TRUE ;
bExec_GearSlaveDyn := FALSE;

// Set feedback Output
CmdGearOut := fbMcGearOutSlave.Done;
END_METHOD

METHOD PUBLIC CmdHalt : BOOL
VAR_INPUT
	fDeceleration 	: LREAL := 0 ; // command deceleration
	mcBuffermode	: MC_BufferMode ; // Buffermode defines how the previous command is executed.
END_VAR
// Set command to true 
bExec_Halt 		:= TRUE ;
bInternalEnable	:= TRUE ;

// coppy parameters
fbMcHalt.Deceleration	:= fDeceleration;
fbMcHalt.BufferMode		:= mcBuffermode	;

// Set feedback output 
CmdHalt := fbMchalt.Active OR fbMcHalt.Done ;
END_METHOD

METHOD PUBLIC CmdHome : BOOL // start axis homing procedure
VAR_INPUT
	fPosition 		: LREAL := 0 ; // Homing position
END_VAR
// set blocked command if halt is active 
bBlockedCommand := fbMcHalt.Active ;

// set command to true 
bExec_Home 		:= TRUE	; 
bInternalEnable	:= TRUE ;

// coppy parameters
fbMcHome.Position 	:= fPosition 	;

// Set feedback output
CmdHome := fbMcHome.Done ;
END_METHOD

METHOD PUBLIC CmdJog : BOOL // Jog axis with variable speed. jog stops as soon as the command is false
VAR_INPUT
	fVelocity		: LREAL 	; // jog velocity can be adjusted as long as the command is active
	fPos			: LREAL 	; // Jog position or step size (if aplicable)
	bJogNegative 	: BOOL 		:= FALSE ; // jog in negative direction
	eJogmode		: E_JogMode := E_JogMode.MC_JOGMODE_CONTINOUS ; // jogmode [default MC_JOGMODE_CONTINOUS] 
END_VAR
// set blocked command if halt is active 
bBlockedCommand := fbMcHalt.Active ;

// Velocity conversion from RPM to deg/sec
	IF bIcfCmdVelocityRpm THEN 
		fVelocity := Rpm_To_DegS(fVelocity);
	END_IF

// Set command to true
	IF fbMcJog.Velocity = fVelocity THEN // If command velocity changes, then set exec to false for one cycle to trigger new velocity so the jog follows the set velocity
		bExec_JogPositive	:= NOT bJogNegative ;
		bExec_JogNegative 	:= bJogNegative ;
	END_IF
	bInternalEnable			:= TRUE ;

// coppy parameters
	fbMcJog.Velocity	:= fVelocity 	;
	fbmcjog.Mode		:= eJogmode		;
	fbMcJog.Position	:= fPos			;

// Set feedback output 
	CmdJog := fbMcJog.Active ;
END_METHOD

METHOD PUBLIC CmdLimitVelocity : BOOL // limit axis maximum velocity, stays active as long as command is called. 
VAR_INPUT
	fVelocityLimit	: LREAL ; // velocity Maximum limit
END_VAR
// set blocked command if halt is active 
bBlockedCommand := fbMcHalt.Active ;

// Set velocity limiting command 
bCmdLimitVelocity S= TRUE;
	
// Set velocity maximum value 
fCmdVelocityLimit := fVelocityLimit ; 

// set feedback 
CmdLimitVelocity := bVelocityLimited ;
END_METHOD

METHOD PUBLIC CmdManual : BOOL
VAR
	eJogmode		: E_JogMode := E_JogMode.MC_JOGMODE_CONTINOUS ; // jogging mode 
END_VAR
// set blocked command if halt is active 
bBlockedCommand := fbMcHalt.Active ;

// Enable axis for manual control
bCmdManual := TRUE ;

// set jog mode 
IF stManualCtrl.bCmdInching THEN 
	eJogmode := E_JogMode.MC_JOGMODE_INCHING ;
END_IF

// execute motion commands
IF stManualCtrl.bCmdJogForward OR stManualCtrl.bCmdJogReverse THEN 
	CmdJog (fVelocity := stManualCtrl.fVelocity, 
			fPos := stManualCtrl.fDistance, 
			bJogNegative := stManualCtrl.bCmdJogReverse, 
			eJogmode := eJogmode);
ELSIF stManualCtrl.bCmdToPos THEN 
	CmdMoveAbs( fPosition := stManualCtrl.fPosition, 
				fVelocity := stManualCtrl.fVelocity, 
				mcBuffermode := MC_BufferMode.MC_Aborting);
ELSIF stManualCtrl.bCmdHome THEN 
	CmdHome( fPosition := 0);
ELSE 
	CmdHalt( 	fDeceleration := fMaxDec * 0.9, 
				mcBuffermode := MC_BufferMode.MC_Aborting) ; 
END_IF
END_METHOD

METHOD PUBLIC CmdMoveAbs : BOOL // Move absolute command
VAR_INPUT
	fPosition	:	LREAL 	; // target position
	fVelocity	: 	LREAL 	; // Maximum velocity [units/sec]
	mcBuffermode: 	MC_BufferMode ; // Buffermode defines how the previous command is executed.
END_VAR
// set blocked command if halt is active 
bBlockedCommand := fbMcHalt.Active ;

// Velocity conversion from RPM to deg/sec
	IF bIcfCmdVelocityRpm THEN 
		fVelocity := Rpm_To_DegS(fVelocity);
	END_IF

// Determine function for command stacking
	IF fbMcMoveAbsolute[0].Active THEN 
		arExec_MoveAbs[1] 				:= (fPosition <> fbMcMoveAbsolute[0].Position OR fVelocity <> fbMcMoveAbsolute[0].Velocity) ;
		fbMcMoveAbsolute[1].Position 	:= fPosition ;
		fbMcMoveAbsolute[1].Velocity 	:= fVelocity ; 
		fbMcMoveAbsolute[1].BufferMode 	:= mcBuffermode ;
	ELSE
		arExec_MoveAbs[0] 				:= (fPosition <> fbMcMoveAbsolute[1].Position OR fVelocity <> fbMcMoveAbsolute[1].Velocity) ;
		fbMcMoveAbsolute[0].Position 	:= fPosition ;
		fbMcMoveAbsolute[0].Velocity 	:= fVelocity ; 
		fbMcMoveAbsolute[0].BufferMode 	:= mcBuffermode ;
	END_IF

bInternalEnable	:= TRUE ;

// set feedback
IF arExec_MoveAbs[1] OR fbMcMoveAbsolute[1].Busy THEN 
	CmdMoveAbs :=	fbMcMoveAbsolute[1].Active ;
ELSE 
	CmdMoveAbs :=	fbMcMoveAbsolute[0].Active ;
END_IF
END_METHOD

METHOD PUBLIC CmdMoveModulo : BOOL // Move to a modulo position
VAR_INPUT
	fPosition	:	LREAL 	; // target position
	fVelocity	: 	LREAL 	; // Maximum velocity [units/sec]
	mcDirection : 	MC_Direction := MC_Direction.MC_Positive_Direction ; // Direction of movement mc_direction [ deafult mc_positive_direction]
	mcBuffermode: 	MC_BufferMode ; // Buffermode defines how the previous command is executed.
END_VAR
// set blocked command if halt is active 
bBlockedCommand := fbMcHalt.Active ;

// Velocity conversion from RPM to deg/sec
	IF bIcfCmdVelocityRpm THEN 
		fVelocity := Rpm_To_DegS(fVelocity);
	END_IF

// Determine function for command stacking
	IF fbMcMoveModulo[0].Active THEN 
		arExec_MoveModulo[1] 		:= (fPosition <> fbMcMoveModulo[0].Position OR fVelocity <> fbMcMoveModulo[0].Velocity)	;
		fbMcMoveModulo[1].Velocity 	:= fVelocity 	;
		fbMcMoveModulo[1].Position 	:= fPosition 	;
		fbMcMoveModulo[1].Direction	:= mcDirection	;
		fbMcMoveModulo[1].BufferMode:= mcBuffermode ;
	ELSE    
		arExec_MoveModulo[0] 		:= (fPosition <> fbMcMoveModulo[1].Position OR fVelocity <> fbMcMoveModulo[1].Velocity) ;
		fbMcMoveModulo[0].Velocity 	:= fVelocity 	;
		fbMcMoveModulo[0].Position 	:= fPosition 	;
		fbMcMoveModulo[0].Direction	:= mcDirection	;
		fbMcMoveModulo[0].BufferMode:= mcBuffermode ;
	END_IF

bInternalEnable	:= TRUE ;

(*// Reset position position and velocity commands
	IF fbMcMoveModulo[1].Active AND NOT fbMcMoveModulo[0].Busy THEN 
		fbMcMoveModulo[0].Velocity := 0 ;
		fbMcMoveModulo[0].Position := 0 ;
	ELSIF fbMcMoveModulo[0].Active AND NOT fbMcMoveModulo[1].Busy THEN 
		fbMcMoveModulo[1].Velocity := 0 ;
		fbMcMoveModulo[1].Position := 0 ;
 	END_IF 
*)
// set feedback
IF arExec_MoveModulo[1] OR fbMcMoveModulo[1].Busy THEN 
	CmdMoveModulo :=	fbMcMoveModulo[1].Active OR fbMcMoveModulo[1].Done;
ELSE
	CmdMoveModulo :=	fbMcMoveModulo[0].Active OR fbMcMoveModulo[0].Done ;
END_IF
END_METHOD

METHOD CmdMoveRelative : BOOL // move relative command 
VAR_INPUT
	fDistance	:	LREAL 	; // target position
	fVelocity	: 	LREAL 	; // Maximum velocity [units/sec]
	mcBuffermode: 	MC_BufferMode ; // Buffermode defines how the previous command is executed.
END_VAR
// set blocked command if halt is active 
bBlockedCommand := fbMcHalt.Active ;

// Velocity conversion from RPM to deg/sec
	IF bIcfCmdVelocityRpm THEN 
		fVelocity := Rpm_To_DegS(fVelocity);
	END_IF

// Determine function for command stacking
	IF fbMCMoveRelative[0].Active THEN 
		arExec_MoveRelative[1] := (fDistance <> fbMCMoveRelative[0].Distance OR fVelocity <> fbMCMoveRelative[0].Velocity) ;
		fbMCMoveRelative[1].Velocity	:= fVelocity 	;
		fbMCMoveRelative[1].Distance	:= fDistance	;
		fbMCMoveRelative[1].BufferMode	:= mcBuffermode	;
	ELSE 
		arExec_MoveRelative[0] := (fDistance <> fbMCMoveRelative[1].Distance OR fVelocity <> fbMCMoveRelative[1].Velocity) ;
		fbMCMoveRelative[0].Velocity	:= fVelocity 	;
		fbMCMoveRelative[0].Distance	:= fDistance	;
		fbMCMoveRelative[0].BufferMode	:= mcBuffermode	;
	END_IF

bInternalEnable	:= TRUE ;

// set feedback
IF arExec_MoveRelative[1] OR fbMCMoveRelative[1].Busy THEN 
	CmdMoveRelative :=	fbMCMoveRelative[1].Active ;
ELSE
	CmdMoveRelative :=	fbMCMoveRelative[0].Active ;
END_IF
END_METHOD

METHOD PUBLIC CmdMoveVelocity : BOOL // Move with set velocity until stopped
VAR_INPUT
	fVelocity	: 	LREAL 	; // Maximum velocity [units/sec]
	mcDirection : 	MC_Direction := MC_Direction.MC_Positive_Direction ; // Direction of movement mc_direction [ deafult mc_positive_direction]
	mcBuffermode: 	MC_BufferMode ; // Buffermode defines how the previous command is executed.
END_VAR
// set blocked command if halt is active 
bBlockedCommand := fbMcHalt.Active ;

// Velocity conversion from RPM to deg/sec
	IF bIcfCmdVelocityRpm THEN 
		fVelocity := Rpm_To_DegS(fVelocity);
	END_IF

// Set command to true 
	bExec_MoveVelocity 	:= TRUE ;
	bInternalEnable		:= TRUE ;

// coppy parameters
	fbMcMoveVelocity.Velocity	:= fVelocity 	;
	fbMcMoveVelocity.Direction 	:= mcDirection	;
	fbMcMoveVelocity.BufferMode	:= mcBuffermode	;

// Set feedback output 
	CmdMoveVelocity := fbMcMoveVelocity.Active ;
END_METHOD

METHOD PUBLIC CmdReset : BOOL
VAR_INPUT
END_VAR
// set blocked command if halt is active 
bBlockedCommand := fbMcHalt.Active ;

// Set reset axis to true 				
	bExec_Reset 	:= TRUE ; 
	bInternalEnable	:= TRUE ;
	
// Set feedback output 
	CmdReset := fbMcReset.Done ;
END_METHOD

METHOD PUBLIC CmdSafeSpeed : BOOL
VAR_INPUT
END_VAR
// Set safestop command
bCmdSafeSpeed := TRUE ; 

// Set feedback output 
CmdSafeSpeed := AxisRef.NcToPlc.ActVelo <= fSafeVeloLimit ;
END_METHOD

METHOD PUBLIC CmdSafeStop : BOOL
VAR_INPUT
END_VAR

// Set safestop command
bCmdSafeStop := TRUE ; 

// Set feedback output 
CmdSafeStop := bDevIsSafe OR NOT bInitOk;
END_METHOD

METHOD PUBLIC Init : BOOL
VAR_INPUT
	// Axis message Data 
	nDevNumber	: UDINT		:= 0	; // Axis number 
	// Config Bits
	bIcfCmdVelocityRpm	: BOOL := FALSE ; // input speeds in Rpm
	bIcfEnableForward 	: BOOL := TRUE 	; // Enable forward motion
	bIcfEnablereverse	: BOOL := TRUE 	; // Enable reverse motion
	bIcfAlwaysEnable	: BOOL := FALSE ; // 1 = Axis always enabled, 0 = Axis disabled at Idle 
	bIcfSimulationMode	: BOOL := FALSE ; // Simulation mode is active [default set to False] Used for testing without hardware present 
	
	// Config Values 
	mcHomingMode 		: MC_HomingMode := MC_HomingMode.MC_DefaultHoming; 
	fHomePosition		: LREAL := 0 	; // set position at homing
	fSafeVeloLimit		: LREAL	:= 360 	; // safe velocity limit [deg/sec]
	nEncTurnoverVal 	: LREAL := 360	; // encoder turnover value 
	tEnableDelay		: time 	:= T#0MS; // Time between axis enable command and motion command execution (0 := no delay active)	
	tDisabledelay		: TIME 	:= T#100MS; // Axis idle time before axis is disabled 
END_VAR
VAR 
	bActVeloReadValid 	: BOOL ; // velocity parameter read is valid 
	bActAccReadValid 	: BOOL ; // Acceleration parameter read is valid 
	bActDecReadValid 	: BOOL ; // Deceleration parameter read is valid 
	bActParamValid 		: BOOL ; // Parameter read is valid 
END_VAR
// Calculate device number
	THIS^.nDevNumber := nDevNumber ;
	SUPER^.CalcDeviceId();

// ===== Message data set =====
	stFault.ComponentType		:= E_ComponentTypes.Axis ;
	
// ===== Read system configuration =====
	McReadSysVelo	(	Axis 			:= AxisRef,
						Enable 			:= Cmd_EnDriveParRead ,
						ParameterNumber := MaxVelocitySystem ,
						ReadMode		:= 1,
						Valid			=> bActVeloReadValid ,						
						Busy			=> ,
						Error			=> ,
						ErrorID			=> ,
						Value			=> fMaxVelo );
	McReadSysAcc	(	Axis 			:= AxisRef,
						Enable 			:= Cmd_EnDriveParRead ,
						ParameterNumber := MaxAccelerationSystem ,
						ReadMode		:= 1,
						Valid			=> bActAccReadValid ,						
						Busy			=> ,
						Error			=> ,
						ErrorID			=> ,
						Value			=> fMaxAcc );
	McReadSysDec	(	Axis 			:= AxisRef,
						Enable 			:= Cmd_EnDriveParRead ,
						ParameterNumber := MaxDecelerationSystem ,
						ReadMode		:= 1,
						Valid			=> bActDecReadValid ,						
						Busy			=> ,
						Error			=> ,
						ErrorID			=> ,
						Value			=> fMaxDec );

	IF 	fMaxVelo > 0 
	AND fMaxAcc >0
	AND fMaxDec >0 THEN 
		bActParamValid	:= TRUE ; 
		fCmdAcc 		:= fMaxAcc * 0.9;
		fCmdDecc		:= fMaxDec * 0.9;
	END_IF

	IF NOT Cmd_EnDriveParRead AND NOT bActParamValid THEN  
		Cmd_EnDriveParRead := TRUE;
	ELSIF Cmd_EnDriveParRead THEN
		Cmd_EnDriveParRead := FALSE;
	END_IF

// ===== Configure Axis =====
	// ***** Config Bits *****
		THIS^.bIcfCmdVelocityRpm	:= bIcfCmdVelocityRpm	; // Enable speed inputs in Rpm
		THIS^.bIcfEnableForward 	:= bIcfEnableForward 	; // Enable forward motion
		THIS^.bIcfEnablereverse		:= bIcfEnablereverse	; // Enable reverse motion
		THIS^.bIcfAlwaysEnable		:= bIcfAlwaysEnable		; // Always enable motor and brake if safety is ok
		THIS^.bIcfSimulationMode	:= bIcfSimulationMode 	; // Simulation mode is active [default set to False] 

	// ***** config homing Mode ***** 
 		THIS^.mcHomingMode 			:= mcHomingMode ; // set homing mode
		THIS^.fHomePosition			:= fHomePosition;
	// ***** Velocity settings *****
		THIS^.fSafeVeloLimit 		:= fSafeVeloLimit ; // set maximum safe velocity	
	// ***** Encoder values *****
		THIS^.fEncoderTurnoverValue := nEncTurnoverVal	; // turnover value for encoder = 25.6 mm per rev * 4096 revolutions 
	// ***** Time delay enable off *****
		THIS^.tEnableDelay		:= tEnableDelay	;
		THIS^.tDisableDelay 	:= tDisabledelay ;		

// ===== Set device type for manual control =====
	eDevType := E_Devices.Axis ;
		
// ===== reset axis state indicators ======
	bError 	:= FALSE;

// ====== Set init to done =======
IF bActParamValid THEN 
	bInitOk	:= TRUE ; 
END_IF
END_METHOD

METHOD INTERNAL ExecGearDynamic : BOOL
VAR_INPUT
END_VAR
// ===== invert gear ratio if reverse slave is active =====
	IF bReverseSlave THEN 
		fbMcGearInDyn.GearRatio := fCmdGearRatio * -1 ;
	ELSE 
		fbMcGearInDyn.GearRatio := fCmdGearRatio ;
	END_IF

// ===== Execute gear in function =====
	fbMcGearInDyn ( 	Master 			:= refMasterAxis,
						Slave			:= AxisRef,
						Enable 			:= bExec_GearSlaveDyn AND bDelayedEnable,
						Acceleration	:= fCmdAcc	); 
						
// ===== reset command =====
	bGearedAsSlave		:= fbMcGearInDyn.InGear ; 

// Gearing fault handling 
	IF fbMcGearInDyn.Error THEN 
		bError					:= TRUE							;
		stFault.Active 			:= TRUE 						;
		stFault.MessageNumber	:= E_MessageNumbers.FF_AxisFault;
		stFault.Discription		:= CONCAT('Gear dynamic Fault ', UDINT_TO_STRING(fbMcGearInDyn.ErrorID));	
		stFault.Discription		:= CONCAT( sDevName , stfault.Discription ) ;
		stFault.FaultType		:= E_FaultTypes.FF				;
		refFbFault.CmdAddFault( stFault );
	END_IF
END_METHOD

METHOD INTERNAL ExecGearIn : BOOL
VAR_INPUT
END_VAR
// ===== invert gear ratio if reverse slave is active =====
	IF bReverseSlave THEN 
		fbMcGearInSlave.RatioNumerator := fCmdGearRatio * -1 ;
	ELSE 
		fbMcGearInSlave.RatioNumerator := fCmdGearRatio ;
	END_IF

// ===== Execute gear in function =====
	fbMcGearInSlave ( 	Master 			:= refMasterAxis,
						Slave			:= AxisRef,
						Execute 		:= bExec_GearAsSlave AND bDelayedEnable,
						RatioDenominator:= 1	); 
						
// ===== reset command =====
	bExec_GearAsSlave 	:= FALSE  ;
	bGearedAsSlave		S= fbMcGearInSlave.InGear ; 

// Gearing fault handling 
	IF fbMcGearInSlave.Error THEN 
		bError					:= TRUE							;
		stFault.Active 			:= TRUE 						;
		stFault.MessageNumber	:= E_MessageNumbers.FF_AxisFault;
		stFault.Discription		:= CONCAT('Gear as slave Fault ', UDINT_TO_STRING(fbMcGearInSlave.ErrorID));
		stFault.Discription		:= CONCAT( sDevName , stfault.Discription ) ;
		stFault.FaultType		:= E_FaultTypes.FF				;
		refFbFault.CmdAddFault( stFault );
	END_IF
END_METHOD

METHOD INTERNAL ExecGearOut : BOOL
VAR_INPUT
END_VAR
// ===== execute gear out function ======
	fbMcGearOutSlave (	Slave 	:= AxisRef,
						Execute := bExec_GearOutSlave );

// ===== reset command =====
	bExec_GearOutSlave	:= false ;
	bGearedAsSlave		R= fbMcGearOutSlave.Done 	; 

// Gearing fault handling 
	IF fbMcGearOutSlave.Error THEN 
		bError					:= TRUE							;
		stFault.Active 			:= TRUE 						;
		stFault.MessageNumber	:= E_MessageNumbers.FF_AxisFault;
		stFault.Discription		:= CONCAT('Gear out Fault ', UDINT_TO_STRING(fbMcGearOutSlave.ErrorID));
		stFault.Discription		:= CONCAT( sDevName , stfault.Discription ) ;
		stFault.FaultType		:= E_FaultTypes.FF				;
		refFbFault.CmdAddFault( stFault );
	END_IF
END_METHOD

METHOD INTERNAL ExecHalt : BOOL
VAR_INPUT
END_VAR
// ==== Execute halt function ===== 
fbMcHalt (	Axis 		:= AxisRef,
			Execute 	:= bExec_Halt );

// ===== reset command =====
	bExec_Halt := FALSE ;
	
// Halt fault handling 
	IF fbMcHalt.Error THEN 
		bError					:= TRUE							;
		stFault.Active 			:= TRUE 						;
		stFault.MessageNumber	:= E_MessageNumbers.FF_AxisFault;
		stFault.Discription		:= CONCAT('Halt Fault ', UDINT_TO_STRING(fbMcHalt.ErrorID));
		stFault.Discription		:= CONCAT( sDevName , stfault.Discription ) ;
		stFault.FaultType		:= E_FaultTypes.FF				;
		refFbFault.CmdAddFault( stFault );
	END_IF
END_METHOD

METHOD INTERNAL ExecHome : BOOL
VAR_INPUT
END_VAR
// ==== execute homing function =====
	fbMcHome(	Axis			:= AxisRef,
				Execute			:= bExec_Home AND bDelayedEnable,
				HomingMode		:= mcHomingMode,
				bCalibrationCam	:= IAxisHome ); 
			
// Reset exec command 
	bExec_Home 	:= FALSE ;
	bHomed		S= fbMcHome.Done ;	
				
// fault handling 
	IF fbMcHome.Error THEN 
		bError					:= TRUE							;
		stFault.Active 			:= TRUE 						;
		stFault.MessageNumber	:= E_MessageNumbers.FF_AxisFault;
		stFault.Discription		:= CONCAT('Homing Fault ', UDINT_TO_STRING(fbMcHome.ErrorID));
		stFault.Discription		:= CONCAT( sDevName , stfault.Discription ) ;
		stFault.FaultType		:= E_FaultTypes.FF				;
		refFbFault.CmdAddFault( stFault );
	END_IF
END_METHOD

METHOD INTERNAL ExecJog : BOOL
VAR_INPUT
END_VAR
// ===== Execute Jog function =====
	// velocity limiting
		IF bCmdSafeSpeed THEN 
			fbMcJog.Velocity := MIN(fSafeVeloLimit, fbMcJog.Velocity); 
		ELSIF bCmdLimitVelocity THEN 
			fbMcJog.Velocity := MIN(fCmdVelocityLimit, fbMcJog.Velocity); 
		END_IF
	// function call
	fbMcJog (	Axis 		:= AxisRef,
				JogForward	:= bExec_JogPositive AND bDelayedEnable,
				JogBackwards:= bExec_JogNegative AND bDelayedEnable,
				Acceleration:= fCmdAcc,
				Deceleration:= fCmdDecc );

// ===== reset command =====
	bExec_JogPositive 	:= FALSE  ;
	bExec_JogNegative	:= FALSE  ;
	
// Jog fault handling 
	IF fbMcJog.Error THEN 
		bError					:= TRUE							;
		stFault.Active 			:= TRUE 						;
		stFault.MessageNumber	:= E_MessageNumbers.FF_AxisFault;
		stFault.Discription		:= CONCAT('Jog Fault ', UDINT_TO_STRING(fbMcJog.ErrorID));
		stFault.Discription		:= CONCAT( sDevName , stfault.Discription ) ;
		stFault.FaultType		:= E_FaultTypes.FF				;
		refFbFault.CmdAddFault( stFault );
	END_IF
END_METHOD

METHOD INTERNAL ExecMoveAbsolute : BOOL
VAR_INPUT
END_VAR
// ==== execute move absolute function =====
FOR i := 0 TO 1 DO 
	// velocity limiting
		IF bCmdSafeSpeed THEN 
			fbMcMoveAbsolute[i].Velocity := MIN(fSafeVeloLimit, fbMcMoveAbsolute[i].Velocity); 
		ELSIF bCmdLimitVelocity THEN 
			fbMcMoveAbsolute[i].Velocity := MIN(fCmdVelocityLimit, fbMcMoveAbsolute[i].Velocity); 
		END_IF
	// function call
	fbMcMoveAbsolute[i](	Axis 		:= AxisRef,
							Execute 	:= arExec_MoveAbs[i] AND bDelayedEnable,
							Acceleration:= fCmdAcc,
							Deceleration:= fCmdDecc );  

	// If function is done then reset command values
	IF fbMcMoveAbsolute[i].Done OR fbMcMoveAbsolute[i].CommandAborted OR NOT arExec_MoveAbs[i] THEN 
		fbMcMoveAbsolute[i].Velocity	:= 0 ;
		fbMcMoveAbsolute[i].Position	:= 0 ; 
	END_IF

	// reset Exec command 
	arExec_MoveAbs[i] := FALSE ; 
	
	// fault handling 
	IF fbMcMoveAbsolute[i].Error THEN 
		bError					:= TRUE							;
		stFault.Active 			:= TRUE 						;
		stFault.MessageNumber	:= E_MessageNumbers.FF_AxisFault;
		stFault.Discription		:= CONCAT('Move absolute Fault ', UDINT_TO_STRING(fbMcMoveAbsolute[i].ErrorID));
		stFault.Discription		:= CONCAT( sDevName , stfault.Discription ) ;
		stFault.FaultType		:= E_FaultTypes.FF				;
		refFbFault.CmdAddFault( stFault );
	END_IF
END_FOR
END_METHOD

METHOD INTERNAL ExecMoveModulo : BOOL
VAR_INPUT
END_VAR
// ===== Execute move modulo function =====
FOR i := 0 TO 1 DO 
	// velocity limiting
		IF bCmdSafeSpeed THEN 
			fbMcMoveModulo[i].Velocity := MIN(fSafeVeloLimit, fbMcMoveModulo[i].Velocity); 
		ELSIF bCmdLimitVelocity THEN 
			fbMcMoveModulo[i].Velocity := MIN(fCmdVelocityLimit, fbMcMoveModulo[i].Velocity); 
		END_IF
	// function call
	fbMcMoveModulo[i](	Axis 		:= AxisRef,
						Execute 	:= arExec_MoveModulo[i] AND bDelayedEnable,
						Acceleration:= fCmdAcc,
						Deceleration:= fCmdDecc);  
	
	// If function is done then reset command values
	IF fbMcMoveModulo[i].Done OR fbMcMoveModulo[i].CommandAborted OR NOT arExec_MoveModulo[i] THEN 
		fbMcMoveModulo[i].Velocity	:= 0 ;
		fbMcMoveModulo[i].Position	:= 0 ; 
	END_IF

	// reset Exec command 
	arExec_MoveModulo[i] := FALSE ; 
	
	// fault handling 
	IF fbMcMoveModulo[i].Error THEN 
		bError					:= TRUE							;
		stFault.Active 			:= TRUE 						;
		stFault.MessageNumber	:= E_MessageNumbers.FF_AxisFault;
		stFault.Discription		:= CONCAT('Move module Fault ', UDINT_TO_STRING(fbMcMoveModulo[i].ErrorID));
		stFault.Discription		:= CONCAT( sDevName , stfault.Discription ) ;
		stFault.FaultType		:= E_FaultTypes.FF			;
		refFbFault.CmdAddFault( stFault );
	END_IF
END_FOR
END_METHOD

METHOD INTERNAL ExecMoveRelative : BOOL
VAR_INPUT
END_VAR
// ===== Execute move relative function ======
FOR i := 0 TO 1 DO 
	// velocity limiting
		IF bCmdSafeSpeed THEN 
			fbMCMoveRelative[i].Velocity := MIN(fSafeVeloLimit, fbMCMoveRelative[i].Velocity); 
		ELSIF bCmdLimitVelocity THEN 
			fbMCMoveRelative[i].Velocity := MIN(fCmdVelocityLimit, fbMCMoveRelative[i].Velocity); 
		END_IF
	// function call
	fbMCMoveRelative[i](	Axis 		:= AxisRef,
							Execute		:= arExec_MoveRelative[i] AND bDelayedEnable,
							Acceleration:= fCmdAcc,
							Deceleration:= fCmdDecc );

	// If function is done then reset command values
	IF fbMCMoveRelative[i].Done OR fbMCMoveRelative[i].CommandAborted OR NOT arExec_MoveRelative[i] THEN 
		fbMCMoveRelative[i].Velocity	:= 0 ;
		fbMCMoveRelative[i].Distance	:= 0 ; 
	END_IF

	// reset Exec command 
	arExec_MoveRelative[i] := FALSE ; 
	
	// fault handling 
	IF fbMCMoveRelative[i].Error THEN 
		bError					:= TRUE							;
		stFault.Active 			:= TRUE 						;
		stFault.MessageNumber	:= E_MessageNumbers.FF_AxisFault;
		stFault.Discription		:= CONCAT('Move relative Fault ', UDINT_TO_STRING(fbMCMoveRelative[i].ErrorID));
		stFault.Discription		:= CONCAT( sDevName , stfault.Discription ) ;
		stFault.FaultType		:= E_FaultTypes.FF			;
		refFbFault.CmdAddFault( stFault );
	END_IF
END_FOR
END_METHOD

METHOD INTERNAL ExecMoveVelocity : BOOL
VAR_INPUT
END_VAR
// ===== Execute move velocity function =====
// velocity limiting
IF bCmdSafeSpeed THEN 
	fbMcMoveVelocity.Velocity := MIN(fSafeVeloLimit, fbMcMoveVelocity.Velocity); 
ELSIF bCmdLimitVelocity THEN 
	fbMcMoveVelocity.Velocity := MIN(fCmdVelocityLimit, fbMcMoveVelocity.Velocity); 
END_IF
// function call
fbMcMoveVelocity (	Axis 		:= AxisRef,
					Execute		:= bExec_MoveVelocity  AND bDelayedEnable,
					Acceleration:= fCmdAcc,
					Deceleration:= fCmdDecc );

// ===== reset command =====
bExec_MoveVelocity := FALSE ;
	
// Halt fault handling 
IF fbMcHalt.Error THEN 
	bError					:= TRUE							;
	stFault.Active 			:= TRUE 						;
	stFault.MessageNumber	:= E_MessageNumbers.FF_AxisFault;
	stFault.Discription		:= CONCAT('Move velocity Fault ', UDINT_TO_STRING(fbMcMoveVelocity.ErrorID));
	stFault.Discription		:= CONCAT( sDevName , stfault.Discription ) ;
	stFault.FaultType		:= E_FaultTypes.FF				;
	refFbFault.CmdAddFault( stFault );
END_IF
END_METHOD

METHOD PRIVATE ExecEnable : BOOL
VAR_INPUT
END_VAR
// ===== Set axis enable ======
IF NOT bEnable AND NOT bCmdManual AND AxisRef.Status.Moving THEN
	CmdHalt(fDeceleration := fCmdDecc, mcBuffermode := MC_BufferMode.MC_Aborting);
ELSE 
	bCmdEnableAxis	:= bEnable OR bCmdManual ;
	bCmdManual := FALSE ;
END_IF

// ===== Check if axis is bussy with a command =====
	bInternalEnable S= AxisRef.Status.HasJob;
	bInternalEnable	S= bIcfAlwaysEnable ; // always enable axis if configured
	bInternalEnable	S= AxisRef.Status.Coupled ;
	
// ===== Axis disable timer after last command =====
	TofIntAxisEnable (	IN:= bInternalEnable, PT := tDisableDelay);

// ===== Enable drive =====
	fbMcPower(	Axis			:= AxisRef , 
				Enable			:= bCmdEnableAxis AND TofIntAxisEnable.Q, 
				Enable_Positive	:= bIcfEnableForward, 
				Enable_Negative	:= bIcfEnablereverse, 
				Override		:= 100 );  
				
// ===== Reset internal enable signal =====
	bInternalEnable := FALSE ; 	

// ===== Delayed enable function =====	
	TonMotionEnable(IN := fbMcPower.Enable, PT := tEnableDelay);
	bDelayedEnable := TonMotionEnable.Q ;	


IF fbMcPower.Error THEN 
	bError					:= TRUE							;
	stFault.Active 			:= TRUE 						;
	stFault.MessageNumber	:= E_MessageNumbers.FF_AxisFault;
	stFault.Discription		:= CONCAT('Enable Fault ', UDINT_TO_STRING(fbMcPower.ErrorID));
	stFault.Discription		:= CONCAT( sDevName , stfault.Discription ) ;
	stFault.FaultType		:= E_FaultTypes.FF				;
	refFbFault.CmdAddFault( stFault );
END_IF
END_METHOD

METHOD INTERNAL ExecReadStatus : BOOL
VAR_INPUT
END_VAR
// Read axis status from drive
fbMcReadAxisStatus (	Enable 	:= TRUE ,
						Axis 	:= AxisRef );
						
// convert velocity to RPM for output if aplicable
IF bIcfCmdVelocityRpm THEN 
	fVelocity := AxisRef.NcToPlc.ActVelo / 6 ;
ELSE 
	fVelocity := AxisRef.NcToPlc.ActVelo ;
END_IF

// write position output
fActPosition := AxisRef.NcToPlc.ActPos ;
						
// set status bits 
bIdle := NOT AxisRef.Status.HasJob ;

// read fault handling 
IF fbMcReadAxisStatus.Error THEN 
	bError					:= TRUE							;
	stFault.Active 			:= TRUE 						;
	stFault.MessageNumber	:= E_MessageNumbers.FF_AxisFault;
	stFault.Discription		:= CONCAT('Status read fault ', UDINT_TO_STRING(fbMcPower.ErrorID));
	stFault.Discription		:= CONCAT( sDevName , stfault.Discription ) ;
	stFault.FaultType		:= E_FaultTypes.FF				;
	refFbFault.CmdAddFault( stFault );
END_IF
END_METHOD

METHOD INTERNAL ExecReset : BOOL
VAR_INPUT
END_VAR
IF  AxisRef.Status.Moving AND bExec_Reset THEN // If the axis is still moving execute safe stop first
	CmdSafeStop();
	RETURN;
END_IF

// ===== Reset axis, drive and axis functions =====
	fbSoeReset ( 	Execute := bExec_Reset AND NOT fbMcReset.Busy AND NOT bIcfSimulationMode, // No physical drive reset necesarry when not connected 
					Timeout := T#10S		,
					Axis	:= AxisRef		);
	
	fbMcReset	( 	Execute	:= bexec_reset AND NOT fbSoeReset.Busy,
					Axis	:= AxisRef ); 
					
// ===== reset command =====
	bExec_Reset := FALSE ;
	
// ===== reset internal fault bits and stop bits =====
	bError 			:= FALSE ; 
	
// Reset fault handling 
	IF fbSoeReset.Error OR fbMcReset.Error THEN 
		bError					:= TRUE							;
		stFault.Active 			:= TRUE 						;
		stFault.MessageNumber	:= E_MessageNumbers.FF_AxisFault;
		stFault.Discription		:= CONCAT('Reset Fault ', UDINT_TO_STRING(fbMcReset.ErrorID));
		stFault.Discription		:= CONCAT( sDevName , stfault.Discription ) ;
		stFault.FaultType		:= E_FaultTypes.FF				;
		refFbFault.CmdAddFault( stFault );
	END_IF
END_METHOD

METHOD PRIVATE ExecSafeFunctions : BOOL
VAR_INPUT
END_VAR
// ==== Stop when safety is not ok =====
	bCmdSafeStop := NOT bSafetyOk ;

// ==== Safe operation functions (overrule all other motion functions) =====
	fbMcStop( 	Axis 			:= AxisRef		,
				Execute 		:= bCmdSafeStop	,
				Deceleration	:= fMaxDec		);
	
	// Reset axis command			
	bCmdSafeStop 	R= fbMcStop.Done OR AxisRef.Status.HasBeenStopped ;
	bStopped		:= AxisRef.Status.HasBeenStopped ;

// Safestop fault handling 
	IF fbMcStop.Error THEN 
		bError					:= TRUE							;
		stFault.Active 			:= TRUE 						;
		stFault.MessageNumber	:= E_MessageNumbers.FF_AxisFault;
		stFault.Discription		:= CONCAT('Safe stop axis fault ', UDINT_TO_STRING(fbMcStop.ErrorID));
		stFault.Discription		:= CONCAT( sDevName , stfault.Discription ) ;
		stFault.FaultType		:= E_FaultTypes.FF				;
		refFbFault.CmdAddFault( stFault );
	END_IF
	
// ===== Safe speed monitoring =====
	IF bCmdSafeSpeed THEN 
		IF AxisRef.NcToPlc.ActVelo > fSafeVeloLimit THEN 
			bExec_Halt := TRUE ; 
			ExecHalt(); 
		ELSE 
			bCmdSafeSpeed := FALSE ; 
		END_IF
	END_IF

// ===== Dev is safe feedback =====
bDevIsSafe := AxisRef.Status.HasBeenStopped AND NOT bCmdEnableAxis  ;
END_METHOD

METHOD PRIVATE CallMotionFunctions : BOOL
VAR_INPUT
END_VAR
// ===== Check if safe to move =====
	IF bCmdSafeStop THEN 
		// ===== reset safe commands ======
		bCmdSafeStop	:= FALSE ; 
		RETURN ;
	END_IF

// ===== Homing functions =====
	ExecHome		(); 

// ===== Motion standstil commands =====
	ExecHalt		();

// ===== Motion move functions
	ExecJog			(); 
	ExecMoveAbsolute();
	ExecMoveRelative();
	ExecMoveModulo	();
	ExecMoveVelocity();
	
// ===== Execute gearing functions =====
	ExecGearIn		();
	ExecGearDynamic	();
	ExecGearOut		();
	
// ====== reset velocity lmiting =====
	bVelocityLimited	:= bCmdLimitVelocity ;	
	bCmdLimitVelocity 	:= FALSE ;
END_METHOD

METHOD PRIVATE CallOrganizationFunctions : BOOL
VAR_INPUT
END_VAR
// ==== execute organizational functions =====
	ExecReadStatus	(); 
	ExecEnable		();
	ExecReset		();
END_METHOD

END_FUNCTION_BLOCK

// Buttons/Functions/FB_DevPushbuttonLight
FUNCTION_BLOCK PUBLIC FB_DevPushbuttonLight EXTENDS Fb_DevDigitalInputFunctions
VAR_OUTPUT
END_VAR
VAR
	fbLight : Fb_DevLight ; // light control 
END_VAR

// Set device type
IF eDevType = E_Devices.Undefined THEN 
	eDevType := E_Devices.PushButtonLight ;
END_IF

SUPER^();

// Light commands
	
fbLight(bEnable := bEnable);

METHOD PUBLIC CmdBlinkFast : BOOL
VAR_INPUT
END_VAR
CmdBlinkFast := fbLight.CmdBlinkFast();
END_METHOD

METHOD PUBLIC CmdBlinkSlow : BOOL
VAR_INPUT
END_VAR
CmdBlinkSlow	:= fbLight.CmdBlinkSlow();
END_METHOD

METHOD PUBLIC CmdOn : BOOL
VAR_INPUT
END_VAR
CmdOn := fbLight.CmdOn() ;
END_METHOD

END_FUNCTION_BLOCK

// Sensors/DigitalSensor/FunctionBlocks/Fb_DevDigitalInputFunctions
FUNCTION_BLOCK PUBLIC Fb_DevDigitalInputFunctions EXTENDS Fb_DevDigitalInput
VAR_OUTPUT
	bFcoDelay			: BOOL			;// Digital sensor, Delayed input status (3 seconds) 
	bFeStatus			: BOOL			;// Digital sensor, Falling edge of input signal	
	bReStatus			: BOOL			;// Digital sensor, Rising edge of input signal
	bFcoFlipFlop		: BOOL			;// Digital sensor, feedback flip flop
	TetInputActive		: TIME			;// Digital sensor, Time elapsed while button is active
END_VAR
VAR
	// ***** Fucntion blocks *****
		FB_delIStatus: TON; // Timer function for delayed input status 
		FB_feIStatus: F_TRIG; // generate falling edge pulse edge from Istatus
		FB_reIStatus: R_TRIG; // generate falling edge pulse edge from Istatus
		FB_rsIStatus: RS; // Set Reset function for flip flop input
END_VAR

SUPER^();

// ====== process functions if enabled ======
	// ***** Set Delayed inputs and time elapsed ****
		FB_delIStatus(	IN:= bFcoInputActive,
						PT:= tDelay , 
						Q=> bFcoDelay , 
						ET=> TetInputActive 
					  ); // Generate delayed input status from push button input status
	// ***** Edge triggers *****
		FB_feIStatus(CLK:= bFcoInputActive , Q=> bFeStatus ); // generate falling edge pulse on pushbutton input
		FB_reIStatus (Clk := bFcoInputActive , Q => bReStatus); // Generate rising edge from push button input signal
	// ***** Flip Flop *****
		FB_rsIStatus(	SET:= bFeStatus AND NOT bFcoFlipFlop , 
						RESET1:= bFeStatus AND bFcoFlipFlop , 
						Q1=> bFcoFlipFlop 
					 ); // Generate set reset function from pushbutton input status

END_FUNCTION_BLOCK

// Sensors/DigitalSensor/FunctionBlocks/Fb_DevDigitalInput
FUNCTION_BLOCK PUBLIC Fb_DevDigitalInput EXTENDS FB_DevBase 
VAR_INPUT
	tDelay			: TIME 	:= T#1S	;// Time before delayed signal becomes active 
	bCmdSimulate	: BOOL 	:= FALSE ;// Simulate sensor Input 
	bSimState		: BOOL 	:= FALSE ;// Simulated sensor state
END_VAR
VAR_OUTPUT
	bFcoInputActive		: BOOL 			;// Digital sensor, Button active state
END_VAR
VAR
	Istatus		AT 	%I* : BOOL			;// Digital sensor, Direct input status
END_VAR

// Set device type
IF eDevType = E_Devices.Undefined THEN 
	eDevType := E_Devices.DigitalSensor ;
END_IF

// Call base function
SUPER^();

// ***** Direct input when enabled *****
IF bEnable THEN 
	IF bCmdSimulate  THEN 
		bFcoInputActive := bSimState ;
		bCmdSimulate	:= FALSE ;  
	ELSE
		bFcoInputActive := Istatus ;
	END_IF
ELSE 
	bFcoInputActive := FALSE ;
END_IF

END_FUNCTION_BLOCK

// Lights/Functions/Fb_DevLight
FUNCTION_BLOCK PUBLIC Fb_DevLight EXTENDS FB_DevBase ;
VAR
	bCmdBlinkSlow	: BOOL := FALSE ; // Command light blink slow
	bCmdBlinkFast 	: BOOL := FALSE ; // Command light blink fast
	bCmdOn			: BOOL := FALSE ; // Command turn light on	 
	qLight AT %Q* 	: BOOL := FALSE ; // light output
END_VAR

// set device type
IF eDevType = E_Devices.Undefined THEN 
	eDevType := E_Devices.DigitalOut ;
END_IF

// ===== check if light is enabled ======
	IF NOT bEnable AND NOT bCmdManual THEN 
		qLight := FALSE ;
		RETURN; 
	END_IF
	
// ===== set light output ======
	ExecSetOutput();

METHOD PRIVATE ExecSetOutput : BOOL
VAR_INPUT
END_VAR
// ===== set light output state =====
IF bCmdOn THEN 
	qLight S= TRUE ;
ELSIF bCmdBlinkFast THEN 
	qLight := Sys_Variables.BlinkFast 	;
ELSIF bCmdBlinkSlow THEN 
	qLight := Sys_Variables.BlinkSlow	;
ELSE
	qLight := FALSE ;
END_IF

// reset all commands 
bCmdOn			:= FALSE ;
bCmdBlinkFast 	:= FALSE ;
bCmdBlinkSlow 	:= FALSE ;
END_METHOD

METHOD PUBLIC CmdBlinkFast : BOOL
VAR_INPUT
END_VAR
bCmdBlinkFast S= TRUE ;

CmdBlinkFast := bCmdBlinkFast ;
END_METHOD

METHOD PUBLIC CmdBlinkSlow : BOOL
VAR_INPUT
END_VAR
bCmdBlinkSlow S= TRUE ;

CmdBlinkSlow	:= bCmdBlinkSlow ;
END_METHOD

METHOD PUBLIC CmdOn : BOOL
VAR_INPUT
END_VAR
bCmdOn S= TRUE ;

CmdOn := qLight ;
END_METHOD

END_FUNCTION_BLOCK

// Sensors/AnalogInput/FunctionBlocks/FB_DevAnalogInput
FUNCTION_BLOCK PUBLIC FB_DevAnalogInput EXTENDS FB_DevBase
VAR_INPUT
	bCmdSimulate	: BOOL 	:= FALSE ;// Simulate sensor Input 
	fSimValue		: INT	:= 0 ;// Simulated sensor state
END_VAR
VAR_OUTPUT
	fValue	: LREAL := 0 ; // Input value from hardware (converted to LREAL)
END_VAR
VAR
	nLimitMin		: INT := Utilities_Library.GVL_FixedValues.nINTMINVALUE ; // Initial value is set to integer minimum value for use with normal def analog inputs 
	nLimitMax 		: INT := Utilities_Library.GVL_FixedValues.nINTMAXVALUE	; // Initial value is set to integer minimum value for use with high def analog inputs
	inHwInput AT%I* : INT ; // Hardware connection
END_VAR

// Set device type
eDevType := E_Devices.AnalogSensor ;

// Call base function
SUPER^();

// set feedback
ExecSetFeedback();

METHOD ExecSetFeedback : BOOL
VAR_INPUT
END_VAR
IF bCmdSimulate THEN 
	fValue := int_to_lreal(fSimValue) ;
ELSE
	fValue := INT_TO_LREAL(inHwInput);
END_IF
END_METHOD

END_FUNCTION_BLOCK

// Outputs/AnalogOutputs/FB_DevAnalogOutput
FUNCTION_BLOCK PUBLIC FB_DevAnalogOutput EXTENDS FB_DevBase 
VAR_INPUT
	fCmdValue		: LREAL := 0 ;
END_VAR
VAR_OUTPUT
	fOutputValue	: LREAL := 0 ;
END_VAR
VAR
	nLimitMin		: INT := -32767 ;
	nLimitMax 		: INT := 32767 ;
	qnHwOut	AT%Q*	: INT := 0 ;
END_VAR

// set device type
IF eDevType = E_Devices.Undefined THEN 
	eDevType := E_Devices.AnalogOut ;
END_IF

// Call base function
SUPER^();

// Call private functions
ExecSetOutput();
ExecSetFeedback();

METHOD INTERNAL ExecSetFeedback : BOOL
VAR_INPUT
END_VAR
// Set feedback 
fOutputValue := INT_TO_LREAL(qnHwOut) ;
END_METHOD

METHOD INTERNAL ExecSetOutput : BOOL
VAR_INPUT
END_VAR
// Set Output to physical device
IF bEnable OR bCmdManual THEN 
	qnHwOut := LREAL_TO_INT(fCmdValue) ; 
	qnHwOut := LIMIT(nLimitMin, qnHwOut, nLimitMax) ; 
ELSE 
	fCmdValue := 0 ; 
END_IF
END_METHOD

END_FUNCTION_BLOCK

// Outputs/DigitalOutputs/FB_DevDigitalOutput
FUNCTION_BLOCK PUBLIC FB_DevDigitalOutput EXTENDS FB_DevBase
VAR_INPUT
	bCmdOn			: BOOL ; // command output status
END_VAR
VAR_OUTPUT
	bOutputState	: BOOL := FALSE ; // State of physical output
END_VAR
VAR
	qbOutput AT%Q* : BOOL ; // Output to physical device
END_VAR

// Call base function
SUPER^();

// Call private functions
ExecSetOutput();
ExecSetFeedback();

METHOD PRIVATE ExecSetFeedback : BOOL
VAR_INPUT
END_VAR
// Set feedback 
bOutputState := qbOutput ;
END_METHOD

METHOD PRIVATE ExecSetOutput : BOOL
VAR_INPUT
END_VAR
// Set Output to physical device
IF bEnable OR bCmdManual THEN 
	qbOutput := bCmdOn ; 
ELSE 
	qbOutput S= FALSE ; 
END_IF
END_METHOD

END_FUNCTION_BLOCK

// Heaters/FB_DevPWMGenerator
FUNCTION_BLOCK PUBLIC FB_DevPWMGenerator EXTENDS FB_DevBase
VAR_INPUT
	nPeriodLength	: DINT	:= 2000 ; // desired PWM cycle time length [ms] 
	nDutyCycle 		: DINT	:= 50 ; // percentage of power [%]
END_VAR
VAR_OUTPUT
END_VAR
VAR
	qbOutput	AT %Q* 	: BOOL 	; // physical output
	bCycleOutput		: BOOL 	; // Cycle output
	tonTimerOn  		: TON 	; // Timer for cycle on
	tofTimerOff			: TOF 	; // timer for cycle off 
	// output commands
	bCmdPWMCycle		: BOOL 	; // run PWM cycle 
	bCmdOn				: BOOL 	; // turn output on permanantly
END_VAR

// Set device type
eDevType := E_Devices.PWMController ;
SUPER^(refFbFault := refFbFault); 

// calculate cycle times 
CalcCycle();
// set outputs
ExecSetOutput(); 

// reset manual enable
bCmdManual := FALSE ;

METHOD PRIVATE CalcCycle : BOOL
VAR_INPUT
END_VAR
// check if dutycycle is within limits
nDutyCycle := LIMIT(1,nDutyCycle,100);

// Calculate time on from cycle time
tonTimerOn.PT 	:= DINT_TO_TIME(( nPeriodLength / 100) * nDutyCycle);
tofTimerOff.PT	:= DINT_TO_TIME(( nPeriodLength / 100) * (100 - nDutyCycle));
END_METHOD

METHOD PRIVATE ExecSetOutput : BOOL
VAR_INPUT
END_VAR

// PWM signal generator
IF bCmdPWMCycle THEN 
	// Run cycle timers 
	tofTimerOff	(IN := tonTimerOn.Q);
	tonTimerOn	(IN := bCycleOutput AND NOT tofTimerOff.Q );
	bCycleOutput := NOT tofTimerOff.Q ;
ELSE
	bCycleOutput := FALSE ;
END_IF

// set output 
IF bSafetyOk AND (bEnable OR bCmdManual) THEN 
	qbOutput := bCycleOutput OR bCmdOn ;
ELSE
	qbOutput := FALSE ;
	RETURN; 
END_IF

// reset continuous on command
bCmdOn := false ;
END_METHOD

METHOD PUBLIC CmdOutputCycle : BOOL // start PWM cycle stays on until off command is given
VAR_INPUT
END_VAR
bCmdPWMCycle 	S= TRUE ;
CmdOutputCycle 	:= bCmdPWMCycle ;
END_METHOD

METHOD PUBLIC CmdOutputOff : BOOL // turn off output signal completely
VAR_INPUT
END_VAR
bCmdPWMCycle 	:= FALSE ;
bCmdOn			:= FALSE ;
CmdOutputOff	:= TRUE 	;
END_METHOD

METHOD PUBLIC CmdOutputOn : BOOL // Output stays on until command ends (returns to PWM if active otherwise turns off)
VAR_INPUT
END_VAR
bCmdOn 		S= TRUE ;
CmdOutputOn	:= TRUE ;
END_METHOD

END_FUNCTION_BLOCK

// Heaters/FB_DevDoublePWM
FUNCTION_BLOCK PUBLIC FB_DevDoublePWM EXTENDS FB_DevBase // PWM control for 2 outputs that cannot be switchid on simultaniously
VAR_INPUT
	bCmdPWMOn			: BOOL := FALSE ; // PWM controller on 
END_VAR
VAR_OUTPUT
END_VAR
VAR
	bCmdChanelAOn		: BOOL := FALSE ; // command switch chanel A on permanently
	bCmdChanelBOn		: BOOL := FALSE ; // Commandswitch chanel B on permanently 
	bCmdOverrulePWM		: BOOL := FALSE ; // Command to overrule PWM
	bCmdHold			: BOOL := false ; // Command hold PWM on signals (collision avoidance)

	tPeriodLength		: TIME  ; // desired PWM cycle time length [ms] 
	tDutyCycle 			: TIME	; // percentage of power [%]
	tIdleTime			: TIME	; // Time both outputs are idle during PWM
	
	tonOutputA 			: TON ; // Timer on PWM output A
	tonOutputB 			: TON ; // Timer on PWM output B
	tonIdle				: TON ; // Timer On PWM Idle time (both outputs off)

	tofOutputA 			: TOF ; // Timer off PWM output A Off (For overlap prevention)
	tofOutputB 			: TOF ; // Timer off PWM output B Off ( for overlap prevention)

	stParPeriodLength	: Udt_Parameter := (fValue := 2000); // desired PWM cycle time length [ms] Parameter
	stParDutyCycle 		: Udt_Parameter	:= ( fValue := 0); // percentage of power [%] Parameter
	stParSwitchOverTime	: Udt_Parameter	; // Time between switching A off and B on (and vice versa) Parameter
	stMaxTimeOn			: Udt_Parameter := (fValue := 1000);// Maximum time a heater can be on without burning through
	
	qbOutputMain AT %Q* 	: BOOL 	; // physical output to main relais
	qbOutputA	 AT %Q* 	: BOOL 	; // physical output to output A
	qbOutputB	 AT %Q* 	: BOOL 	; // physical output to output B
	
	nPWMStep	: INT ; // PWM stepper

	tonBurnTimeA	: TON ; // burn timer for coil A
	tonBurnTimeB	: TON ; // burn timer for coil B 
END_VAR

// set device type
IF eDevType = E_Devices.Undefined THEN 
	eDevType := E_Devices.DoublePWMController ;
END_IF

// Call base function
SUPER^();

// ===== hold all actions if not initialized ======
IF NOT bInitOk THEN
	RETURN;
END_IF 

// call Functions 
CalcCycleTimes();
IF tDutyCycle > T#0S AND tPeriodLength > T#0S THEN // switch PWM controller up when cycle timer is null
	ExecPWMCycle(); // 
END_IF 

SetOutputs();

METHOD INTERNAL CalcCycleTimes : BOOL // calculate cycle timers
VAR_INPUT
END_VAR
VAR 
END_VAR
// Calculate Cycle timers
tPeriodLength	:= LREAL_TO_TIME( stParPeriodLength.fValue );
tDutyCycle		:= LREAL_TO_TIME(stParPeriodLength.fValue * (stParDutyCycle.fValue / 100));
tIdleTime		:= LREAL_TO_TIME(stParPeriodLength.fValue) - (tDutyCycle * 2) ;

tofOutputA.PT := LREAL_TO_TIME(stParSwitchOverTime.fValue);
tofOutputB.PT := LREAL_TO_TIME(stParSwitchOverTime.fValue);
END_METHOD

METHOD INTERNAL ExecPWMCycle : BOOL
VAR_INPUT
END_VAR
IF bCmdPWMOn THEN 
	IF bCmdOverrulePWM OR bCmdHold THEN 
		IF bCmdChanelAOn THEN 
			nPWMStep := 1 ;
		ELSE 
			nPWMStep := 0 ;
		END_IF
		bCmdOverrulePWM := FALSE ;
		RETURN;
	END_IF
ELSE 
	RETURN;
END_IF

// PWM stepper 
CASE nPWMStep OF 
	0: // Switch on chanel A
		bCmdChanelAOn := TRUE ;
		IF tonOutputA.Q THEN
			nPWMStep := 1 ;
		END_IF
	1: // Switch on chanel B
		bCmdChanelBOn := TRUE;
		IF tonOutputB.Q THEN
			nPWMStep := 2 ;
		END_IF
	2: // Idle Time 
		IF tonIdle.Q THEN 
			nPWMStep := 0;
		END_IF
	ELSE
		;
END_CASE

// call timers 
tonOutputA	(IN := bCmdChanelAOn, PT := tDutyCycle);
tonOutputB	(IN := bCmdChanelBOn, PT := tDutyCycle);
tonIdle 	(IN := nPWMStep = 2	, PT := tIdleTime);
END_METHOD

METHOD PRIVATE SetOutputs : BOOL
VAR_INPUT
END_VAR

// Set main output
qbOutputMain := (bEnable OR bManual) AND bSafetyOk AND NOT bCmdHold ;

// Set outputs
qbOutputA := bCmdChanelAOn AND NOT tofOutputB.Q AND NOT tonBurnTimeA.Q;
qbOutputB := bCmdChanelBOn AND NOT tofOutputA.Q AND NOT tonBurnTimeB.Q;

// Call timers for overlap prevention
tofOutputA(IN := qbOutputA);
tofOutputB(IN := qbOutputB);

// reset commands
bCmdChanelAOn := FALSE ;
bCmdChanelBOn := FALSE ;

tonBurnTimeA ( IN := bCmdChanelAOn, PT := LREAL_TO_TIME( stMaxTimeOn.fValue));
tonBurnTimeB ( IN := bCmdChanelBOn, PT := LREAL_TO_TIME( stMaxTimeOn.fValue));

IF tonBurnTimeA.Q THEN 
	stFault.Active 			:= TRUE ;
	stFault.Discription 	:= 'Heater A burn timeout';
	stFault.MessageNumber 	:= E_MessageNumbers.CF_MoveToSlow ;
	stFault.FaultType		:= E_FaultTypes.CF;
	qbOutputA 				:= FALSE ;
ELSIF tonBurnTimeB.Q THEN 
	stFault.Active 			:= TRUE ;
	stFault.Discription 	:= 'Heater B burn timeout';
	stFault.MessageNumber 	:= E_MessageNumbers.CF_MoveToSlow ;
	stFault.FaultType		:= E_FaultTypes.CF;
	qbOutputB 				:= FALSE ;
END_IF

bCmdHold := FALSE ;
END_METHOD

METHOD PUBLIC CmdHold : BOOL
VAR_INPUT
END_VAR
bCmdHold := TRUE ;

CmdHold := NOT qbOutputMain ;
END_METHOD

METHOD PUBLIC CmdOutputAOn : BOOL // Turn on chanel A permanently 
VAR_INPUT
END_VAR
bCmdOverrulePWM S= TRUE ;
bCmdChanelAOn S= TRUE ;

CmdOutputAOn := qbOutputA AND qbOutputMain ;
END_METHOD

METHOD PUBLIC CmdOutputBOn : BOOL
VAR_INPUT
END_VAR
bCmdOverrulePWM S= TRUE ;
bCmdChanelBOn S= TRUE ;

CmdOutputBOn := qbOutputB AND qbOutputMain ;
END_METHOD

METHOD PUBLIC CmdSafeStop : BOOL
VAR_INPUT
END_VAR
bCmdOverrulePWM S= TRUE ;
bCmdChanelAOn 		:= FALSE ;
bCmdChanelBOn		:= FALSE ;
qbOutputMain 		:= FALSE ;

bDevIsSafe := NOT (qbOutputA OR qbOutputB OR qbOutputMain);
END_METHOD

METHOD PUBLIC Init : BOOL
VAR_INPUT
	nDevNumber		: UDINT	:= 0	; // Cylinder identification number
END_VAR
// ====== Calculate device id =====
	THIS^.nDevNumber := nDevNumber ;
	SUPER^.CalcDeviceId();
// ====== Set message information =======
	stFault.ComponentType	:= E_ComponentTypes.Heaters	;

// ======= Reset Error bit ======
	bErrorActive 	:= FALSE;
	bBussy			:= FALSE;
	
// ===== configure parameters =====
	stParPeriodLength.fMinimum 		:= 0 		;
	stParPeriodLength.fMaximum		:= 60000 	;
	stParPeriodLength.nNumber 		:= nDevId + 1;
	stParPeriodLength.sDiscription  := CONCAT( STR1 := sDevName, STR2 := 'Period length of the cycle in miliseconds');
	stParPeriodLength.sName			:= CONCAT( STR1 := sDevName, STR2 := 'Period Length');
	stParPeriodLength.sType			:= 'MPar';
	stParPeriodLength.sUnit			:= 'ms';
	stParPeriodLength.fValue		:= 5000;

	stParDutyCycle.fMinimum 		:= 0 		;
	stParDutyCycle.fMaximum			:= 50 		;
	stParDutyCycle.nNumber 			:= nDevId + 2;
	stParDutyCycle.sDiscription  	:= CONCAT( STR1 := sDevName, STR2 := 'Percentage of period length in which an output is active');
	stParDutyCycle.sName			:= CONCAT( STR1 := sDevName, STR2 := 'Duty Cyle');
	stParDutyCycle.sType			:= 'MPar';
	stParDutyCycle.sUnit			:= '%';
	stParPeriodLength.fValue		:= 10;

	
	stParSwitchOverTime.fMinimum 	:= 0 		;
	stParSwitchOverTime.fMaximum	:= 500 		;
	stParSwitchOverTime.nNumber 	:= nDevId + 3;
	stParSwitchOverTime.sDiscription:= CONCAT( STR1 := sDevName, STR2 := 'Idle time between output chanel switchover in miliseconds');
	stParSwitchOverTime.sName		:= CONCAT( STR1 := sDevName, STR2 := 'Switch Time');
	stParSwitchOverTime.sType		:= 'CPar';
	stParSwitchOverTime.sUnit		:= 'ms';

	stMaxTimeOn.fMinimum 	:= 0 		;
	stMaxTimeOn.fMaximum	:= 5000 	;
	stMaxTimeOn.nNumber 	:= nDevId + 4;
	stMaxTimeOn.sDiscription:= CONCAT( STR1 := sDevName, STR2 := 'Maximum time a heater can be fully on without burning through');
	stMaxTimeOn.sName		:= CONCAT( STR1 := sDevName, STR2 := 'Max heating time');
	stMaxTimeOn.sType		:= 'MPar';
	stMaxTimeOn.sUnit		:= 'ms';
	
	
	// add parameters to handler 
	refFbParHandler.CmdAddParameter( refParameter := stParPeriodLength );
	refFbParHandler.CmdAddParameter( refParameter := stParDutyCycle );
	refFbParHandler.CmdAddParameter( refParameter := stParSwitchOverTime );
	
// ====== Set init status bit =======
	bInitOk := TRUE ;
END_METHOD

END_FUNCTION_BLOCK

// Actuators/Cylinder/MLTFunctions/Fb_DevSupportCyl
FUNCTION_BLOCK PUBLIC Fb_DevSupportCyl EXTENDS Fb_DevCylWithFbk
VAR_INPUT
	// Traverse data
	stTraverseAxisRef	: AXIS_REF 			; // Axis reference
	nHandCartPos		: LREAL 			; // Position of hand cart
	tMindownTime		: TIME	:= T#1S		; // minimum time down before it can go up again 
END_VAR
VAR_OUTPUT
	bStopAll			: BOOL := TRUE 	; // Support fault stop all motions 
	// feedback 
	bSupportOk			: BOOL := FALSE 	; // Support is running ok
	 
END_VAR
VAR
	bCmdSupportDown		: BOOL 	:= FALSE 	; // External command to move support down 
	// Support data
	nSupportPosition	: LREAL := 0 		; // possition of support cylinder in reference to the home position 
	nSupportWidth		: LREAL := 100		; // width of support cylinder 
	// Traverse data 
	nTravMaxAcc				: LREAL ; // traverse maximum acceleration 
	nTravMaxDec				: LREAL ; // traverse maximum deceleration 
	nTraverseLength			: LREAL	:= 550		; // Length of sewing head Traverse 
	nTraverseFlagPosition	: LREAL	:= 0		; // position of flag in reference to edge of Traverse 
	
	// handcart data
	nHandCartLength			: LREAL := 100	; // Length of hand cart 
	nHandCartClearance		: LREAL := 300	; // Clearance around cart in which support is down
	
	// safety values 	
	nMinSafeDistanceDown: LREAL := 200	; // Minimum distance for support to move down

	// Traverse triggers 
	nMinStopDistance 	: 	LREAL 	:= 10		; // Minimum stopping distance required[mm]
	nTriggerDown		: 	LREAL	:= 100		; // trigger distance for support to go down[mm]
	nTriggerUp			: 	LREAL	:= 50 		; // trigger distance for support to move up[mm]
	nTriggerPosDownFw	:	LREAL 	; // trigger position for support to move down when moving forward [mm]
	nTriggerPosCheckDownFw: LREAL 	; // trigger for safety check is cylinder is down when mocing forward [mm]
	nTriggerPosDownRe	: 	LREAL 	; // trigger position for support to move down when moving reverse [mm]
	nTriggerPosCheckDownRe: LREAL 	; // trigger for safety check is cylinder is down when mocing reverse [mm]

	nTriggerPosUpFw		: 	LREAL	; // Trigger position for support to move Up [mm]
	nTriggerPosUprev	: 	LREAL	; // Trigger position for support to move Up [mm]
	
	// handcart down positions
	nCartCmdDownHigh	: LREAL ; // hand cart position for cylinder to go down high limit
	nCartCmdDownLow		: LREAL ; // hand cart Position for cylinder to go down low limit 
	
	fbTimerStartup		:	TON		; // Startup time before support down check
	
	// Support down trigger
	bSupportClose 	: BOOL 	; // Support close command
	tonSupportDown 	: TON 	; // support Down command
	
END_VAR

IF NOT bInitOk THEN
	bStopAll	:= TRUE ; 
	RETURN;
ELSE
	;
END_IF 

// ======= Enable/ disable support cylinder dependent functions =======
	bStopAll := bErrorActive OR bCmdManual OR NOT bEnable ; 	

// ======= Activate cylinder ======	
SUPER^(refFbFault := refFbFault);

// ====== Manual functions =====
	IF bCmdManual THEN 
		bCmdManual		:= FALSE ;	
		RETURN;
	END_IF
	
// ======= Calculate variables =======
	ExecCalc();	

// ======= Support cylinder control =======
	IF bCmdSupportDown THEN 
		CmdClose();
		IF bFco_Closed THEN 
			bCmdSupportDown := FALSE ;
		END_IF
 	ELSE
		ExecCylControl();
	END_IF

METHOD PROTECTED ExecCalc : BOOL
VAR_INPUT
END_VAR
VAR 
	nTriggerOffset 	: LREAL ;
	nMaxAccelDist	: LREAL ;
	nMaxVelocity	: LREAL ;
	nDecelDist		: LREAL	;
	nTraverseFront		: LREAL ; // front of Traverse distance from sensor flag
END_VAR
// ***** Calculate hardstop distance *****
	nMinStopDistance	:= (ABS(stTraverseAxisRef.NcToPlc.ActVelo) / 2) * (ABS(stTraverseAxisRef.NcToPlc.ActVelo) / nTravMaxDec);
	
// ***** Calculate speed dependant trigger offset *****
	nTriggerOffset := F_TriggerPosOffset( Velocity := ABS(stTraverseAxisRef.NcToPlc.ActVelo), nMoveTimeMs := stTimesClose.Maximum);

// ***** Calculate triggerdistance down *****
	nTriggerDown := (nSupportWidth / 2) + nMinStopDistance + nTriggerOffset;
	IF nTriggerDown < nMinSafeDistanceDown THEN 
		nTriggerDown := nMinSafeDistanceDown ;
	END_IF
	
// ***** Calculate triggerdistance Up *****
	nMaxAccelDist 	:= F_AccDecDistanceFromTime	(nAccelDecel:= nTravMaxAcc, nTimeMs := stTimesClose.Maximum);
	nMaxVelocity	:= F_TopVelocityFromTime	(nAccel 	:= nTravMaxAcc, nTimeMs := stTimesClose.Maximum);
	nDecelDist		:= F_AccDecDistanceFromVelo (nAccDecc	:= nTravMaxDec, nVelocity := nMaxVelocity);
	
	nTriggerUp	:= ((nSupportWidth / 2) + nMaxAccelDist + nDecelDist)* 1.1; // 1.1 is a %10 safety margint to account for cycle time 


// ***** calculate traverse lenght from sensor *****
	nTraverseFront := nTraverseLength - nTraverseFlagPosition ;

	
// ===== Calculate trigger positions =====
	// ***** positive direction positions *****
		nTriggerPosDownFw		:= nSupportPosition - nTriggerDown - nTraverseFront ;
		nTriggerPosCheckDownFw	:= nSupportPosition - (nSupportWidth / 2) - nTraverseFront - nMinStopDistance ; 
		nTriggerPosUpFw			:= nSupportPosition + nTraverseFlagPosition + nTriggerUp;
		
	// ***** negative direction positions *****
		nTriggerPosDownRe 		:= nSupportPosition + nTriggerDown + nTraverseFlagPosition ;
		nTriggerPosCheckDownRe	:= nSupportPosition + (nSupportWidth / 2) + nTraverseFlagPosition + nMinStopDistance; 
		nTriggerPosUprev		:= nSupportPosition - nTraverseFront - nTriggerUp;
	
// ===== calculate hand cart trigger positions ======
	nCartCmdDownHigh 	:= nSupportPosition + nHandCartClearance ;
	nCartCmdDownLow		:= nSupportPosition - nHandCartClearance - nHandCartLength  ;
END_METHOD

METHOD PROTECTED ExecCylControl : BOOL
VAR
	nTravPos : LREAL ;
END_VAR
// ===== copy position in temporary var (for readability ) ======
	nTravPos := stTraverseAxisRef.NcToPlc.ActPos ; 

// ===== Trigger Support cylinder =====
	IF nHandCartPos >= nCartCmdDownLow AND nHandCartPos <= nCartCmdDownHigh THEN  
		bSupportClose := TRUE ;
	ELSIF 	stTraverseAxisRef.Status.PositiveDirection 
		AND	nTravPos >= nTriggerPosDownFw 
		AND nTravPos <= nTriggerPosUpFw 
		THEN 
		bSupportClose := TRUE ;
	ELSIF 	stTraverseAxisRef.Status.NegativeDirection  
		AND nTravPos <= nTriggerPosDownRe 
		AND nTravPos >= nTriggerPosUprev 
		THEN 
		bSupportClose := TRUE ;
	ELSIF	nTravPos > nTriggerPosUprev AND nTravPos < nTriggerPosUpFw THEN 
		bSupportClose := TRUE ;
	ELSE
		bSupportClose := FALSE ;
	END_IF

// ===== Run filter timer =====
	tonSupportDown(IN := bFco_Closed, PT := tMindownTime);	

// ===== Set Cylinder command ======
	IF bSupportClose THEN 
		CmdClose() ;
	ELSIF tonSupportDown.Q THEN 
		CmdOpen();
	END_IF
END_METHOD

